PROPERTY xMoverPathFree : BOOL
GET
xMoverPathFree := THIS^.fb_Pnp.xOUT_MoverFree OR THIS^.fb_Pnp.xOUT_Ready OR THIS^.fb_Pnp.xOUT_Done;
END_GET
END_PROPERTY

PROPERTY xMoverShouldLeave : BOOL
GET
xMoverShouldLeave := THIS^.fb_Pnp.iOUT_Step = ST120_Pnp_e.SYNC_MOVER_LEAVE;
END_GET
END_PROPERTY

END_FUNCTION_BLOCK

// ---- POUs/20_AUTO/ST120/FB_ABL_120_Pnp.TcPOU
FUNCTION_BLOCK FB_ABL_120_Pnp
(****************************************************************************************)
(*	TITEL				laden kristall- Modul	    										*)
(*	Status				ungetestet                         								*)
(*	Beschrieb:			Ablaufbeschreibung												*)
(*																						*)
(*	Steps:	self-explained using enum													*)
(***********************************Revisionen*******************************************)
(*	see github blames																	*)
(****************************************************************************************)

VAR_INPUT
    xIN_Reset       : BOOL;          // Schrittkette zurücksetzen 
    xIN_Init        : BOOL;          // Initialisieren
    xIN_Quit        : BOOL;          // Fehler quittieren 
    xIN_Start       : BOOL;          // Startbefehl
    xIN_Sperre      : BOOL;          // FB Sperren 
    xIN_NextStep    : BOOL;          // Nächsten Schritt ausführen 
    xIN_AlarmAktiv  : BOOL;          // Anlage hat Alarm
    xIN_DryCycle    : BOOL;          // Fahren ohne Teile
    xIN_RestartCYCL : BOOL;          // Zyklus erneut starten im STEP, END, LEERFAHREN
    enIN_State      : enState;       // Status Anlage
    tIN_Timeout     : TIME := T#10s; // Timout

    pxFG_Freigabe : POINTER TO BOOL; //Freigabe von Station

    // Application specific
    Mover              : REFERENCE TO FB_Mover;
    xIN_PceReadyToPick : BOOL; // the piece(s) is/are ready to picked
END_VAR
VAR_OUTPUT
    (* standart Ausgänge *)
    xOUT_ErrFlag  : BOOL;        // Error Flag 
    xOUT_Busy     : BOOL;        // Baustein befindet sich im Ablauf 
    xOUT_Done     : BOOL;        // Baustein hat den Ablauf beendet 		
    xOUT_Ready    : BOOL;        // Ready to begin, should be the same state as done	
    xOUT_Timeout  : BOOL;        // Timeout FB 
    xOUT_InitDone : BOOL;        // initialisierung fertig
    xOUT_Wait     : BOOL;        // Wartet auf Bedingung
    iOUT_Step     : ST120_Pnp_e; // Aktueller Schritt 
    sOUT_Step     : STRING;      // Aktueller Schritt but in string format
    bOUT_Error    : BYTE;        // Fehlernummer

    iOUT_ProcessCompletion : INT;  //process completion, express in % (0-100)
    xOUT_MoverFree         : BOOL; // The mover is free to move
    xOUT_PickPiece         : BOOL; // Set to true when a piece is picked

END_VAR
VAR
    (* Standard *)
    (* Schritt *)
    iLastStep : ST120_Pnp_e; // Merker letzter Schritt 
    iPreStep  : ST120_Pnp_e; // Schritt zurück nach Alarm 
    iAktStep  : ST120_Pnp_e; // aktueller Schritt

    // Trigger Starten 
    rtSTART : R_TRIG;
    // Timer TimeOut 
    TON_Timeout : TON;

    (* Bausteine *)

    (* Spezial *)
    fb_axis120_01Y : FB_AxisLM_V1_1;
    fb_axis120_02Z : FB_AxisLM_V1_1;

    fb_PnpHorAxis : FB_LinearMotionMan;
    fb_PnpVerAxis : FB_LinearMotionMan;

    fb_gripperLeft    : FB_ZylMo2El_V2_1;
    fb_gripperRight   : FB_ZylMo2El_V2_1;
    simu_gripperLeft  : FB_Simu_Zyl2Pos;
    simu_gripperRight : FB_Simu_Zyl2Pos;

    fb_simu_axis120_01Y : FB_Simu_AxisLM_V1_1;
    fb_simu_axis120_02Z : FB_Simu_AxisLM_V1_1;

END_VAR
VAR CONSTANT
    PNP_SIMULATION : BOOL := FALSE; // Set to TRUE to simulate this part of the program
END_VAR

(*******************************************************************)
(* Trigger  *)
(*******************************************************************)
(* Zurücksetzen *)
IF xIN_RESET THEN
    iPreStep  := ST120_Pnp_e.RESET;
    iOUT_Step := ST120_Pnp_e.RESET;
END_IF

(* Error Quittieren *)
IF (bOUT_Error <> 0) AND xIN_Quit THEN
    xOUT_ErrFlag := FALSE;
    bOUT_Error   := 0;
    iOUT_Step    := iPreStep;
END_IF

(*******************************************************************)
(* Timer *)
(*******************************************************************)
TON_Timeout(IN := xIN_NextStep AND (iLastStep = iOUT_Step) (*todo FG *) ,
            PT := tIN_Timeout);

(*******************************************************************)
(* Bausteine *)
(*******************************************************************)
fb_PnpHorAxis(config          := _20_AUTO.recipe.linearAxis[LinearAxis_e.ST120_01Y],
              xIN_Init        := enIN_State = enState.StateINIT,
              xIN_Reset       := xIN_Reset,
              lrIN_CurrPos    := fb_axis120_01Y.rOUT_ActPos,
              lrIN_Delta_mm   := 0.5,
              iIN_CurrentStep := iOUT_Step,
              iIN_moveNumber  := ST120_PnpHorPos_e._max);

fb_simu_axis120_01Y(xIN_Enable          := PNP_SIMULATION AND CONST.USE_SIMULATION,
                    bIN_AxisCntr        := fb_axis120_01Y.bOUT_AxisCntr,
                    wIN_AxisState       := ST120_Axis.axis120_01Y.wState,
                    udiIN_HomingTime_ms := 2000,
                    pIN_axisSimu        := ADR(SIMU.axis_ref[Axis_e.ST120_01Y]),
                    pIN_axisHW          := ADR(ST120_Axis.axis120_01Y.axis),
                    rIN_PosActual       := fb_axis120_01Y.rOUT_ActPos,
                    rIN_PosMax          := ST120_Axis.const120_01Y.POS_MAX,
                    rIN_PosMin          := ST120_Axis.const120_01Y.POS_MIN,
                    rIN_PixMax          := 100,
                    rIN_PixMin          := 0);

fb_axis120_01Y(enIN_State       := enIN_State,
               parIN_Buttons    := ADR(AXIS.btTeachArAxis[Axis_e.ST120_01Y]),
               xIN_DisButtons   :=,
               xIN_Quit         := xIN_Quit,
               xIN_PARAMok      := TRUE, (*TODO*)
               xIN_FREE         := TRUE,
               xIN_FREE_HOME    := TRUE,
               rIN_POSMIN       := ST120_Axis.const120_01Y.POS_MIN,
               rIN_POSMAX       := ST120_Axis.const120_01Y.POS_MAX,
               rIN_VELOMAX      := ST120_Axis.const120_01Y.VELO_MAX,
               rIN_VELOMANU     := ST120_Axis.const120_01Y.VELO_MANU,
               rIN_VELOOPEN     := ST120_Axis.const120_01Y.VELO_MANU / 4,
               rIN_JogInc       := AXIS.rTeachIncAxis,
               xIN_Execute      := fb_PnpHorAxis.xOUT_Execute,
               xIN_Home         := ST120_Pnp_e.Init_HomeHorizontals = iAktStep,
               xIN_Relative     :=,
               rIN_Position     := TO_REAL(fb_PnpHorAxis.OUT_MoveProfile.lrPosition),
               rIN_Velocity     := TO_REAL(fb_PnpHorAxis.OUT_MoveProfile.lrVelocity),
               rIN_Acceleration := TO_REAL(fb_PnpHorAxis.OUT_MoveProfile.lrAccel),
               rIN_Deceleration := TO_REAL(fb_PnpHorAxis.OUT_MoveProfile.lrDecel),
               rIN_Jerk         := TO_REAL(fb_PnpHorAxis.OUT_MoveProfile.lrJerk),
               rIN_PosManu      :=
               TO_REAL(_20_AUTO.recipe
                           .linearAxis[LinearAxis_e.ST120_01Y].movesList[AXIS.bTeachPos[Axis_e.ST120_01Y]].lrPosition),
               rIN_VeloJogManu := TO_REAL(Axis.rJogVelo_pc),
               xIN_Reset       := (ST120_Pnp_e.RESET = iAktStep) OR xIN_Reset,
               // the simu fb gives the hardware signal when the simulation is disabled
               wAxisState    := fb_simu_axis120_01Y.wOUT_AxisState,
               bOUT_AxisCntr => ST120_Axis.axis120_01Y.bCtrlHi,
               rOUT_ActPos   => ST120_Axis.axis120_01Y.rActPos,
               axisIN_REF    := fb_simu_axis120_01Y.pOUT_axisRef^);

fb_PnpVerAxis(config          := _20_AUTO.recipe.linearAxis[LinearAxis_e.ST120_02Z],
              xIN_Init        := enIN_State = enState.StateINIT,
              xIN_Reset       := xIN_Reset,
              lrIN_CurrPos    := fb_axis120_02Z.rOUT_ActPos,
              lrIN_Delta_mm   := 0.5,
              iIN_CurrentStep := iOUT_Step,
              iIN_moveNumber  := ST120_PnpVerPos_e._max);

fb_simu_axis120_02Z(xIN_Enable          := PNP_SIMULATION AND CONST.USE_SIMULATION,
                    bIN_AxisCntr        := fb_axis120_02Z.bOUT_AxisCntr,
                    wIN_AxisState       := ST120_Axis.axis120_02Z.wState,
                    udiIN_HomingTime_ms := 2000,
                    pIN_axisSimu        := ADR(SIMU.axis_ref[Axis_e.ST120_02Z]),
                    pIN_axisHW          := ADR(ST120_Axis.axis120_02Z.axis),
                    rIN_PosActual       := fb_axis120_02Z.rOUT_ActPos,
                    rIN_PosMax          := ST120_Axis.const120_02Z.POS_MAX,
                    rIN_PosMin          := ST120_Axis.const120_02Z.POS_MIN,
                    rIN_PixMax          := 100,
                    rIN_PixMin          := 0);

fb_axis120_02Z(enIN_State       := enIN_State,
               parIN_Buttons    := ADR(AXIS.btTeachArAxis[Axis_e.ST120_02Z]),
               xIN_DisButtons   :=,
               xIN_Quit         := xIN_Quit,
               xIN_PARAMok      := TRUE, (*TODO*)
               xIN_FREE         := TRUE,
               xIN_FREE_HOME    := TRUE,
               rIN_POSMIN       := ST120_Axis.const120_02Z.POS_MIN,
               rIN_POSMAX       := ST120_Axis.const120_02Z.POS_MAX,
               rIN_VELOMAX      := ST120_Axis.const120_02Z.VELO_MAX,
               rIN_VELOMANU     := ST120_Axis.const120_02Z.VELO_MANU,
               rIN_VELOOPEN     := ST120_Axis.const120_02Z.VELO_MANU / 4,
               rIN_JogInc       := AXIS.rTeachIncAxis,
               xIN_Execute      := fb_PnpVerAxis.xOUT_Execute,
               xIN_Home         := ST120_Pnp_e.Init_HomeVerticals = iAktStep,
               xIN_Relative     :=,
               rIN_Position     := TO_REAL(fb_PnpVerAxis.OUT_MoveProfile.lrPosition),
               rIN_Velocity     := TO_REAL(fb_PnpVerAxis.OUT_MoveProfile.lrVelocity),
               rIN_Acceleration := TO_REAL(fb_PnpVerAxis.OUT_MoveProfile.lrAccel),
               rIN_Deceleration := TO_REAL(fb_PnpVerAxis.OUT_MoveProfile.lrDecel),
               rIN_Jerk         := TO_REAL(fb_PnpVerAxis.OUT_MoveProfile.lrJerk),
               rIN_PosManu      :=
               TO_REAL(_20_AUTO.recipe
                           .linearAxis[LinearAxis_e.ST120_02Z].movesList[AXIS.bTeachPos[Axis_e.ST120_02Z]].lrPosition),
               rIN_VeloJogManu := TO_REAL(Axis.rJogVelo_pc),
               xIN_Reset       := (ST120_Pnp_e.RESET = iAktStep) OR xIN_Reset,
               // the simu fb gives the hardware signal when the simulation is disabled
               wAxisState    := fb_simu_axis120_02Z.wOUT_AxisState,
               bOUT_AxisCntr => ST120_Axis.axis120_02Z.bCtrlHi,
               rOUT_ActPos   => ST120_Axis.axis120_02Z.rActPos,
               axisIN_REF    := fb_simu_axis120_02Z.pOUT_axisRef^);

fb_gripperLeft(xIN_Reset    := xIN_Reset OR (ST120_Pnp_e.RESET = iOUT_Step),
               xIN_Quit     := xIN_Quit,
               xIN_Manu     := enState.StateMANU = enIN_State,
               pbtIN_Button := ADR(HMI.btManuCylinders[StationList_e.ST120][1]),
               xIN_GS       := simu_gripperLeft.xOUT_inGS,
               xIN_AS       := simu_gripperLeft.xOUT_inAS,
               xIN_FREE     := TRUE,
               xINtoGS      := (ST120_Pnp_e.Gripper_open = iOUT_Step) OR
                               (ST120_Pnp_e.Init_open_left_clamp = iOUT_Step),
               xINtoAS      := _20_AUTO.recipe.st120.xUseVerLeft AND ST120_Pnp_e.Gripper_close = iOUT_Step,
               tIN_ErrAS := DINT_TO_TIME(_20_AUTO.recipe.cylinder2Pos[StationList_e.ST120]
                                             [ST120_Cylinders_e.GreiferLinks].toAS_alarm_time),
               tIN_ErrGS := DINT_TO_TIME(_20_AUTO.recipe.cylinder2Pos[StationList_e.ST120]
                                             [ST120_Cylinders_e.GreiferLinks].toGS_alarm_time),
               tIN_WaitAS := DINT_TO_TIME(_20_AUTO.recipe.cylinder2Pos[StationList_e.ST120]
                                              [ST120_Cylinders_e.GreiferLinks].toAS_wait_time),
               tIN_WaitGS := DINT_TO_TIME(_20_AUTO.recipe.cylinder2Pos[StationList_e.ST120]
                                              [ST120_Cylinders_e.GreiferLinks].toGS_wait_time));

simu_gripperLeft(xIN_Enable := TRUE, // PNP_SIMULATION AND CONST.USE_SIMULATION,
                 xIN_inGS   := IO_BOX.I6300_ST120_greifer_links_geschlossen,
                 xIN_inAS   := IO_BOX.I6301_ST120_greifer_links_offen,
                 xIN_valve  := fb_gripperLeft.xOUT_VALVE,
                 tIN_GS_ms  := 200,  //ms
                 tIN_AS_ms  := 200); //ms

fb_gripperRight(xIN_Reset    := xIN_Reset OR (ST120_Pnp_e.RESET = iOUT_Step),
                xIN_Quit     := xIN_Quit,
                xIN_Manu     := enState.StateMANU = enIN_State,
                pbtIN_Button := ADR(HMI.btManuCylinders[StationList_e.ST120][2]),
                xIN_GS       := simu_gripperRight.xOUT_inGS,
                xIN_AS       := simu_gripperRight.xOUT_inAS,
                xIN_FREE     := TRUE,
                xINtoGS      := (ST120_Pnp_e.Gripper_open = iOUT_Step) OR
                                (ST120_Pnp_e.Init_open_right_clamp = iOUT_Step),
                xINtoAS      := _20_AUTO.recipe.st120.xUseVerRight AND (ST120_Pnp_e.Gripper_close = iOUT_Step),
                tIN_ErrAS := DINT_TO_TIME(_20_AUTO.recipe.cylinder2Pos[StationList_e.ST120]
                                              [ST120_Cylinders_e.GreiferRechts].toAS_alarm_time),
                tIN_ErrGS := DINT_TO_TIME(_20_AUTO.recipe.cylinder2Pos[StationList_e.ST120]
                                              [ST120_Cylinders_e.GreiferRechts].toGS_alarm_time),
                tIN_WaitAS := DINT_TO_TIME(_20_AUTO.recipe.cylinder2Pos[StationList_e.ST120]
                                               [ST120_Cylinders_e.GreiferRechts].toAS_wait_time),
                tIN_WaitGS := DINT_TO_TIME(_20_AUTO.recipe.cylinder2Pos[StationList_e.ST120]
                                               [ST120_Cylinders_e.GreiferRechts].toGS_wait_time));

simu_gripperRight(xIN_Enable := TRUE, // PNP_SIMULATION AND CONST.USE_SIMULATION,
                  xIN_inGS   := IO_BOX.I6302_ST120_greifer_rechts_geschlossen,
                  xIN_inAS   := IO_BOX.I6303_ST120_greifer_rechts_offen,
                  xIN_valve  := fb_gripperRight.xOUT_VALVE,
                  tIN_GS_ms  := 200,  //ms
                  tIN_AS_ms  := 200); //ms

(*******************************************************************)
(* OUTPUTS *)
(*******************************************************************)
// Error Flag 
xOUT_ErrFlag := (bOUT_Error <> 0) OR (ST120_Pnp_e.ERROR = iOUT_Step);
// Baustein befindet sich im Ablauf 
xOUT_Busy := (iOUT_Step > ST120_Pnp_e.READY) AND (iOUT_Step < ST120_Pnp_e.DONE);
// Baustein hat den Ablauf beendet
xOUT_Done := (iOUT_Step = ST120_Pnp_e.DONE);
// Process ready
xOUT_Ready := (iOUT_Step = ST120_Pnp_e.READY) OR (iOUT_Step = ST120_Pnp_e.waitOnMover);
// Timeout FB 				 		
xOUT_Timeout := TON_Timeout.Q;
// Itialisierung fertig			
xOUT_InitDone := (iOUT_Step = ST120_Pnp_e.READY) OR (iOUT_Step = ST120_Pnp_e.waitOnMover);
// Aktueller Schritt			
iOUT_Step := iOUT_Step; //Im Ablauf gesetzt		
sOUT_Step := TO_STRING(iOUT_Step);
//Fehlernummer	 
bOUT_Error := bOUT_Error; //Im Ablauf/FB gesetzt	
(* Warte (alle Schritte wo auf FG oder Teile gewartet wird) *)
xOUT_Wait := (iOUT_Step = ST120_Pnp_e.DONE) OR
             (iOUT_Step = ST120_Pnp_e.READY) OR
             (iOUT_Step = ST120_Pnp_e.START) OR
             (iOUT_Step = ST120_Pnp_e.waitOnMover) OR
             (iOUT_Step = ST120_Pnp_e.SYNC_MOVER_LEAVE) OR
             (iOUT_Step = ST120_Pnp_e.PnP_WaitOnFeeder);

xOUT_MoverFree := iOUT_Step >= ST120_Pnp_e.MOVER_FREE_OP AND iOUT_Step < ST120_Pnp_e.MOVER_NEEDED_OP;

iOUT_ProcessCompletion := F_GetPercent_2(iAktStep,
                                         ST120_Pnp_e.PnP_Hor_ToRotTablePos,
                                         ST120_Pnp_e.PnP_Hor_ToTrackPos,
                                         ST120_Pnp_e.PnP_Ver_ShuttleDown,
                                         ST120_Pnp_e.PnP_Ver_ShuttleUp);

xOUT_PickPiece := iOUT_Step = ST120_Pnp_e.PnP_Ver_RotTableUp;

IO_BOX.Q5202_14_ST120_greifer_links  := fb_gripperLeft.xOUT_VALVE AND NOT (PNP_SIMULATION AND CONST.USE_SIMULATION);
IO_BOX.Q5203_14_ST120_greifer_rechts := fb_gripperRight.xOUT_VALVE AND NOT (PNP_SIMULATION AND CONST.USE_SIMULATION);

IO_BOX.Q5212_14_ST120_stop_vertical_axis := NOT fb_simu_axis120_02Z.pIN_axisHW^.Status.Error AND
                                            _02_SAFETY.xOUT_ESout AND
                                            _02_SAFETY.xOUT_MonOut AND
                                            NOT (PNP_SIMULATION AND CONST.USE_SIMULATION);

(*******************************************************************)
(* Ablauf *)
(*******************************************************************)

(* Sperren *)
IF xIN_Sperre THEN
    iPreStep  := ST120_Pnp_e.RESET;
    iOUT_Step := ST120_Pnp_e.RESET;
    RETURN;
END_IF;

(* Schritt Merker *)
IF iAktStep <> iOUT_Step THEN
    iLastStep := iAktStep;
    iAktStep  := iOUT_Step;
END_IF

(* START *)
rtSTART(CLK := xIN_Start);

IF 0 = bOUT_Error THEN
    IF fb_axis120_01Y.xOUT_ErrFlag THEN
        bOUT_Error := ST120_Alarm_e.Axis_120_01Y_error;
    ELSIF fb_axis120_02Z.xOUT_ErrFlag THEN
        bOUT_Error := ST120_Alarm_e.Axis_120_02Z_error;
    ELSIF fb_gripperLeft.xOUT_ErrFlag THEN
        bOUT_Error := ST120_Alarm_e.Cylinder_griper_left;
    ELSIF fb_gripperRight.xOUT_ErrFlag THEN
        bOUT_Error := ST120_Alarm_e.Cylinder_griper_right;
    END_IF
ELSIF iOUT_Step < ST120_Pnp_e.ERROR THEN
    iOUT_Step := ST120_Pnp_e.ERROR;
END_IF

(*******************************************************************)
(* Schrittkette  *)
(*******************************************************************)
CASE iOUT_Step OF

(***** RESET *****)
ST120_Pnp_e.RESET: (* Schritt 0-99 *)
    //Initialisierungen
    //Start Init Ablauf
    IF xIN_Init THEN
        iOUT_Step := ST120_Pnp_e.INIT;
        //Start Manu Ablauf
    ELSIF enIN_State = StateMANU AND xIN_NextStep THEN
        iOUT_Step := ST120_Pnp_e.INIT;
    END_IF;

(***** INIT *****)
ST120_Pnp_e.INIT: (* Grundstellung ? *)
    IF fb_axis120_02Z.xOUT_HOMED THEN
        iOUT_Step := ST120_Pnp_e.Init_VerticalsUp;
    ELSE
        iOUT_Step := ST120_Pnp_e.Init_HomeVerticals;
    END_IF

ST120_Pnp_e.Init_HomeVerticals:
    IF fb_axis120_02Z.xOUT_HOMED THEN
        iOUT_Step := ST120_Pnp_e.Init_VerticalsUp;
    END_IF

ST120_Pnp_e.Init_VerticalsUp:
    IF fb_gripperLeft.xIN_AS OR fb_gripperRight.xIN_AS THEN
        IF fb_PnpVerAxis.MoveTo(ST120_PnpVerPos_e.UpFull).xOUT_InPos THEN
            IF fb_axis120_01Y.xOUT_READY OR fb_axis120_01Y.xOUT_HOMED THEN
                iOUT_Step := ST120_Pnp_e.Init_HorizontalsToTrack;
            ELSE
                iOUT_Step := ST120_Pnp_e.Init_HomeHorizontals;
            END_IF
        END_IF
    ELSE
        IF fb_PnpVerAxis.MoveTo(ST120_PnpVerPos_e.UpEmpty).xOUT_InPos THEN
            IF fb_axis120_01Y.xOUT_READY OR fb_axis120_01Y.xOUT_HOMED THEN
                iOUT_Step := ST120_Pnp_e.Init_HorizontalsToTrack;
            ELSE
                iOUT_Step := ST120_Pnp_e.Init_HomeHorizontals;
            END_IF
        END_IF
    END_IF

ST120_Pnp_e.Init_HomeHorizontals:
    IF fb_axis120_01Y.xOUT_HOMED THEN
        iOUT_Step := ST120_Pnp_e.Init_HorizontalsToTrack;
    END_IF

ST120_Pnp_e.Init_HorizontalsToTrack:
    IF fb_PnpHorAxis.MoveTo(ST120_PnpHorPos_e.GS).xOUT_InPos THEN
        iOUT_Step := ST120_Pnp_e.Init_adjust_left_clamp;
    END_IF

ST120_Pnp_e.Init_adjust_left_clamp:
    // a piece is in the griper when there is no GS signal
    IF _20_AUTO.recipe.st120.xUseVerLeft THEN
        iOUT_Step := ST120_Pnp_e.Init_adjust_right_clamp;
    ELSE
        iOUT_Step := ST120_Pnp_e.Init_open_left_clamp;
    END_IF

ST120_Pnp_e.Init_open_left_clamp:
    IF fb_gripperLeft.xIN_GS THEN
        IF _20_AUTO.recipe.st120.xUseVerRight THEN
            iOUT_Step := ST120_Pnp_e.Init_adjust_right_clamp;
        ELSE
            iOUT_Step := ST120_Pnp_e.Init_check_if_pces_handled;
        END_IF
    END_IF

ST120_Pnp_e.Init_adjust_right_clamp:
    // a piece is in the griper when there is no GS signal
    IF _20_AUTO.recipe.st120.xUseVerRight THEN
        iOUT_Step := ST120_Pnp_e.Init_check_if_pces_handled;
    ELSE
        iOUT_Step := ST120_Pnp_e.Init_open_right_clamp;
    END_IF

ST120_Pnp_e.Init_open_right_clamp:
    IF fb_gripperRight.xIN_GS THEN
        iOUT_Step := ST120_Pnp_e.Init_check_if_pces_handled;
    END_IF

ST120_Pnp_e.Init_check_if_pces_handled:
    IF (NOT _20_AUTO.recipe.st120.xUseVerLeft AND NOT fb_gripperLeft.xIN_GS) OR
       (NOT _20_AUTO.recipe.st120.xUseVerRight AND NOT fb_gripperRight.xIN_GS) THEN
        bOUT_Error := ST120_Alarm_e.Piece_in_unused_griper;
        iOUT_Step  := ST120_Pnp_e.ERROR;

    ELSIF (_20_AUTO.recipe.st120.xUseVerLeft AND fb_gripperLeft.xIN_GS) AND
          (_20_AUTO.recipe.st120.xUseVerRight AND NOT fb_gripperRight.xIN_GS) THEN
        bOUT_Error := ST120_Alarm_e.Piece_missing_left_griper;
        iOUT_Step  := ST120_Pnp_e.ERROR;

    ELSIF (_20_AUTO.recipe.st120.xUseVerLeft AND NOT fb_gripperLeft.xIN_GS) AND
          (_20_AUTO.recipe.st120.xUseVerRight AND fb_gripperRight.xIN_GS) THEN
        bOUT_Error := ST120_Alarm_e.Piece_missing_right_griper;
        iOUT_Step  := ST120_Pnp_e.ERROR;

        // if both are open, we don't make further checks
    ELSIF (NOT _20_AUTO.recipe.st120.xUseVerLeft OR fb_gripperLeft.xOUT_inGS) AND
          (NOT _20_AUTO.recipe.st120.xUseVerRight OR fb_gripperRight.xOUT_inGS) THEN
        iOUT_Step := ST120_Pnp_e.waitOnMover;

    ELSE
        iOUT_Step := ST120_Pnp_e.READY;
    END_IF

(***** READY / INIT DONE *****)
ST120_Pnp_e.READY:    (* Start AUTO,END,LEER,STEP *)
    IF xIN_Start THEN //IF rtSTART.Q THEN
        iOUT_Step := ST120_Pnp_e.START;
    END_IF

(***** START  ZYKLISCH *****)
ST120_Pnp_e.START: (*  *)
    IF xIN_NextStep AND pxFG_Freigabe^ THEN
        IF enState.StateLEER = enIN_State THEN
            IF __ISVALIDREF(Mover) THEN
                IF Mover.GetLastStationDone() > 0 THEN
                    iOUT_Step := ST120_Pnp_e.PnP_Hor_ToRotTablePos;
                ELSE
                    iOUT_Step := ST120_Pnp_e.waitOnMover;
                END_IF
            END_IF
        ELSE
            iOUT_Step := ST120_Pnp_e.PnP_Hor_ToRotTablePos;
        END_IF
    END_IF;

ST120_Pnp_e.PnP_Hor_ToRotTablePos:
    IF xIN_NextStep AND fb_PnpHorAxis.MoveTo(ST120_PnpHorPos_e.AS).xOUT_InPos THEN
        iOUT_Step := ST120_Pnp_e.PnP_WaitOnFeeder;
    END_IF

ST120_Pnp_e.PnP_WaitOnFeeder:
    IF xIN_PceReadyToPick THEN
        iOUT_Step := ST120_Pnp_e.PnP_Ver_RotTableDown;
    END_IF

ST120_Pnp_e.PnP_Ver_RotTableDown:
    IF xIN_NextStep AND fb_PnpVerAxis.MoveTo(ST120_PnpVerPos_e.DownEmpty).xOUT_InPos THEN
        iOUT_Step := ST120_Pnp_e.Gripper_close;
    END_IF;

ST120_Pnp_e.Gripper_close:
    IF xIN_NextStep AND
       (NOT _20_AUTO.recipe.st120.xUseVerLeft OR fb_gripperLeft.xOUT_inAS) AND
       (NOT _20_AUTO.recipe.st120.xUseVerRight OR fb_gripperRight.xOUT_inAS) THEN
        iOUT_Step := ST120_Pnp_e.PnP_Ver_RotTableUp;
    END_IF;

ST120_Pnp_e.PnP_Ver_RotTableUp:
    IF xIN_NextStep AND fb_PnpVerAxis.MoveTo(ST120_PnpVerPos_e.UpFull).xOUT_InPos THEN
        iOUT_Step := ST120_Pnp_e.PnP_Hor_ToTrackPos;
    END_IF;

ST120_Pnp_e.PnP_Hor_ToTrackPos:
    IF xIN_NextStep AND fb_PnpHorAxis.MoveTo(ST120_PnpHorPos_e.GS).xOUT_InPos THEN
        iOUT_Step := ST120_Pnp_e.waitOnMover;
    END_IF

ST120_Pnp_e.waitOnMover: (*  *)
    IF xIN_NextStep AND __ISVALIDREF(Mover) OR HMI.bArForceCyclusState[StationList_e.ST120] THEN
        IF Mover.GetLastStationDone() >= INT#120 THEN
            iOUT_Step := ST120_Pnp_e.SYNC_MOVER_LEAVE;
        ELSIF Mover.GetLastStationDone() < INT#105 THEN
            iOUT_Step := ST120_Pnp_e.SYNC_MOVER_LEAVE;
        ELSE
            iOUT_Step := ST120_Pnp_e.PnP_Ver_ShuttleDown;
        END_IF
    END_IF;

ST120_Pnp_e.PnP_Ver_ShuttleDown:
    IF xIN_NextStep AND fb_PnpVerAxis.MoveTo(ST120_PnpVerPos_e.DownFullQuick).xOUT_InPos THEN
        iOUT_Step := ST120_Pnp_e.PnP_Ver_ShuttleTorqueControl;

        IF __ISVALIDREF(Mover) THEN
            IF NOT Mover.SetLastStation(120) THEN
                ASSERT(0);
            END_IF
        END_IF
    END_IF;

// We need a fb that enables for us torque control. Here we just go a bit further
ST120_Pnp_e.PnP_Ver_ShuttleTorqueControl:
    IF xIN_NextStep AND fb_PnpVerAxis.MoveTo(ST120_PnpVerPos_e.DownFullTorqueControl).xOUT_InPos THEN
        iOUT_Step := ST120_Pnp_e.Gripper_open;
    END_IF;

ST120_Pnp_e.Gripper_open:
    IF xIN_NextStep AND
       (NOT _20_AUTO.recipe.st120.xUseVerLeft OR fb_gripperLeft.xOUT_inGS) AND
       (NOT _20_AUTO.recipe.st120.xUseVerRight OR fb_gripperRight.xOUT_inGS) THEN
        iOUT_Step := ST120_Pnp_e.PnP_Ver_ShuttleUp;
    END_IF;

ST120_Pnp_e.PnP_Ver_ShuttleUp:
    IF xIN_NextStep AND fb_PnpVerAxis.MoveTo(ST120_PnpVerPos_e.UpEmpty).xOUT_InPos THEN
        iOUT_Step := ST120_Pnp_e.SYNC_MOVER_LEAVE;

        IF __ISVALIDREF(Mover) THEN
            IF NOT Mover.SetLastStation(120) THEN
                ASSERT(0);
            END_IF
        END_IF
    END_IF;

ST120_Pnp_e.SYNC_MOVER_LEAVE:
    // The mover needs to be taken by MoverMan
    IF NOT __ISVALIDREF(Mover) THEN
        IF (NOT _20_AUTO.recipe.st120.xUseVerLeft OR fb_gripperLeft.xOUT_inGS AND
           (NOT _20_AUTO.recipe.st120.xUseVerRight OR fb_gripperRight.xOUT_inGS) THEN
            iOUT_Step := ST120_Pnp_e.DONE;
        ELSE
            iOUT_Step := ST120_Pnp_e.waitOnMover;
        END_IF
    END_IF

(***** DONE *****)
ST120_Pnp_e.DONE: (* Letzter Schritt  *)
    IF NOT xIN_AlarmAktiv THEN
        //AUTO
        IF (enIN_State = StateAUTO) AND xIN_RestartCYCL THEN
            iOUT_Step := ST120_Pnp_e.START;
            //STEP / END / LEERFAHREN restart
        ELSIF (enIN_State < StateAUTO) AND (enIN_State >= enState.StateSTEP) AND xIN_RestartCYCL THEN
            iOUT_Step := ST120_Pnp_e.START;
            //STEP / END / LEERFAHREN fertig
        ELSIF (enIN_State = StateREADY) THEN
            iOUT_Step := ST120_Pnp_e.READY;
        END_IF;
    END_IF;

(************ ERROR *************)
ST120_Pnp_e.ERROR: (* ERROR *) ;

END_CASE;

END_FUNCTION_BLOCK

// ---- POUs/20_AUTO/ST120/FB_ABL_120_Feeder.TcPOU
FUNCTION_BLOCK FB_ABL_120_Feeder
(****************************************************************************************)
(*	TITEL				laden Kristall modul, Feeder and rotary table                   *)
(*	Status				ungetestet                         								*)
(*	Beschrieb:			Ablaufbeschreibung												*)
(*																						*)
(*	Steps:	self-explained using enum													*)
(***********************************Revisionen*******************************************)
(*	see github blames																	*)
(****************************************************************************************)

VAR_INPUT
    xIN_Reset       : BOOL;          // Schrittkette zurücksetzen 
    xIN_Init        : BOOL;          // Initialisieren
    xIN_Quit        : BOOL;          // Fehler quittieren 
    xIN_Start       : BOOL;          // Startbefehl
    xIN_Sperre      : BOOL;          // FB Sperren 
    xIN_NextStep    : BOOL;          // Nächsten Schritt ausführen 
    xIN_AlarmAktiv  : BOOL;          // Anlage hat Alarm
    xIN_DryCycle    : BOOL;          // Fahren ohne Teile
    xIN_RestartCYCL : BOOL;          // Zyklus erneut starten im STEP, END, LEERFAHREN
    enIN_State      : enState;       // Status Anlage
    tIN_Timeout     : TIME := T#10s; // Timout

    pxFG_Freigabe : POINTER TO BOOL; //Freigabe von Station

    // Application specific
    xIN_PickPiece : BOOL; (* signal from the pick and place element
                             the number of picked signal depend on the recipe *)
    xIN_PnpGripperOpen : BOOL; // the gripper of the pnp part is open
    xIN_PnpNotOnTheWay : BOOL; // the pnp is at the track side or up enough
END_VAR
VAR_OUTPUT
    (* standart Ausgänge *)
    xOUT_ErrFlag  : BOOL;           // Error Flag 
    xOUT_Busy     : BOOL;           // Baustein befindet sich im Ablauf 
    xOUT_Done     : BOOL;           // Baustein hat den Ablauf beendet 		
    xOUT_Ready    : BOOL;           // Ready to begin, should be the same state as done	
    xOUT_Timeout  : BOOL;           // Timeout FB 
    xOUT_InitDone : BOOL;           // initialisierung fertig
    xOUT_Wait     : BOOL;           // Wartet auf Bedingung
    iOUT_Step     : ST120_Feeder_e; // Aktueller Schritt 
    sOUT_Step     : STRING;         // Aktueller Schritt but in string format
    bOUT_Error    : BYTE;           // Fehlernummer

    // Application specific
    xOUT_PceReadyToPick : BOOL; // the piece(s) is/are ready to picked
END_VAR
VAR
    (* Standard *)
    (* Schritt *)
    iLastStep : ST120_Feeder_e; // Merker letzter Schritt 
    iPreStep  : ST120_Feeder_e; // Schritt zurück nach Alarm 
    iAktStep  : ST120_Feeder_e; // aktueller Schritt

    // Trigger Starten 
    rtSTART : R_TRIG;
    // Timer TimeOut 
    TON_Timeout : TON;

    (* Bausteine *)
	btfb_feederLeft					: FB_BUTTON;
	btfb_feederRight				: FB_BUTTON;

    // Application specific^
    fb_pivotLeft    : FB_ZylMo2El_V2_1;
    fb_pivotRight   : FB_ZylMo2El_V2_1;
    simu_pivotLeft  : FB_Simu_Zyl2Pos;
    simu_pivotRight : FB_Simu_Zyl2Pos;

    simu_feederLeft  : FB_Simu_Feeder;                    // simulation of a feeder
    simu_feederRight : FB_Simu_Feeder;                    // simulation of a feeder
    simu_fifoLeft    : FB_Fifo(BAND_SIZE_FOR_TUBE_LEFT);  // fifo to hold a piece
    simu_fifoRight   : FB_Fifo(BAND_SIZE_FOR_TUBE_RIGHT); // fifo to hold a piece
    rtPutPieceLeft   : R_TRIG;                            // trigger to add a piece
    rtPutPieceRight  : R_TRIG;                            // trigger to add a piece

    fb_feederLeft      : FB_Feeder2Sensors;
    fb_feederRight     : FB_Feeder2Sensors;
    fb_hubladerLeft    : FB_ZylMo2El_V2_1;
    fb_hubladerRight   : FB_ZylMo2El_V2_1;
    simu_hubladerLeft  : FB_Simu_Zyl2Pos;
    simu_hubladerRight : FB_Simu_Zyl2Pos;

    simu_start_tick : UDINT; // simulation start tick, used to simulate movement

    TON_PieceInPivotLeft  : TON;
    TON_PieceInPivotRight : TON;

END_VAR
VAR CONSTANT
    BAND_SIZE_FOR_TUBE_LEFT  : INT := 3; // Band size, we assume that tubes pushe each other in order to move to the PNP machine
    BAND_SIZE_FOR_TUBE_RIGHT : INT := 2; // Band size, we assume that tubes pushe each other in order to move to the PNP machine

    FEEDER_SIMULATION : BOOL := FALSE; // Simulate this code
END_VAR

(*******************************************************************)
(* Trigger  *)
(*******************************************************************)
(* Zurücksetzen *)
IF xIN_RESET THEN
    iPreStep  := ST120_Feeder_e.RESET;
    iOUT_Step := ST120_Feeder_e.RESET;
END_IF;

(* Error Quittieren *)
IF (bOUT_Error <> 0) AND xIN_Quit THEN
    xOUT_ErrFlag := FALSE;
    bOUT_Error   := 0;
    iOUT_Step    := iPreStep;
END_IF;

(*******************************************************************)
(* Timer *)
(*******************************************************************)
TON_Timeout(IN := xIN_NextStep AND (iLastStep = iOUT_Step) (*todo FG *) ,
            PT := tIN_Timeout);

TON_PieceInPivotLeft(IN := IO_BOX.I6404_ST120_teil_in_vereizelung_links,
                     PT := DINT_TO_TIME(_20_AUTO.recipe.st120.TON_PieceInSeperatorLeft));

TON_PieceInPivotRight(IN := IO_BOX.I6405_ST120_teil_in_vereinzelung_rechts,
                      PT := DINT_TO_TIME(_20_AUTO.recipe.st120.TON_PieceInSeperatorRight));

(*******************************************************************)
(* Bausteine *)
(*******************************************************************)
fb_pivotLeft(xIN_Reset    := xIN_Reset OR (ST120_Feeder_e.RESET = iOUT_Step),
             xIN_Quit     := xIN_Quit,
             xIN_Manu     := enState.StateMANU = enIN_State,
             pbtIN_Button := ADR(HMI.btManuCylinders[StationList_e.ST120][3]),
             xIN_GS       := simu_pivotLeft.xOUT_inGS,
             xIN_AS       := simu_pivotLeft.xOUT_inAS,
             xIN_FREE     := xIN_PnpNotOnTheWay OR xIN_PnpGripperOpen,
             xINtoGS      :=
                 _20_AUTO.recipe.st120.xUseVerLeft AND
                 ((ST120_Feeder_e.rotate_to_pnp = iOUT_Step) OR (ST120_Feeder_e.Init_pivot_to_pnp = iOUT_Step)),
             xINtoAS := _20_AUTO.recipe.st120.xUseVerLeft AND
                        (ST120_Feeder_e.rotate_to_feeder = iOUT_Step OR
                        ST120_Feeder_e.Init_pivot_to_feeder = iOUT_Step),
             tIN_ErrAS := DINT_TO_TIME(_20_AUTO.recipe.cylinder2Pos[StationList_e.ST120]
                                           [ST120_Cylinders_e.GreiferLinks].toAS_alarm_time),
             tIN_ErrGS := DINT_TO_TIME(_20_AUTO.recipe.cylinder2Pos[StationList_e.ST120]
                                           [ST120_Cylinders_e.GreiferLinks].toGS_alarm_time),
             tIN_WaitAS := DINT_TO_TIME(_20_AUTO.recipe.cylinder2Pos[StationList_e.ST120]
                                            [ST120_Cylinders_e.GreiferLinks].toAS_wait_time),
             tIN_WaitGS := DINT_TO_TIME(_20_AUTO.recipe.cylinder2Pos[StationList_e.ST120]
                                            [ST120_Cylinders_e.GreiferLinks].toGS_wait_time));

simu_pivotLeft(xIN_Enable := FEEDER_SIMULATION AND CONST.USE_SIMULATION,
               xIN_inGS   := IO_BOX.I6400_ST120_schwenken_links_in_vertikal,
               xIN_inAS   := IO_BOX.I6401_ST120_schwenken_links_in_horizontal,
               xIN_valve  := fb_pivotLeft.xOUT_VALVE,
               tIN_GS_ms  := 500,  //ms
               tIN_AS_ms  := 500); //ms

fb_pivotRight(xIN_Reset    := xIN_Reset OR (ST120_Feeder_e.RESET = iOUT_Step),
              xIN_Quit     := xIN_Quit,
              xIN_Manu     := enState.StateMANU = enIN_State,
              pbtIN_Button := ADR(HMI.btManuCylinders[StationList_e.ST120][4]),
              xIN_GS       := simu_pivotRight.xOUT_inGS,
              xIN_AS       := simu_pivotRight.xOUT_inAS,
              xIN_FREE     := xIN_PnpGripperOpen OR xIN_PnpNotOnTheWay,
              xINtoGS      :=
                  _20_AUTO.recipe.st120.xUseVerRight AND
                  ((ST120_Feeder_e.rotate_to_pnp = iOUT_Step) OR (ST120_Feeder_e.Init_pivot_to_pnp = iOUT_Step)),
              xINtoAS := _20_AUTO.recipe.st120.xUseVerRight AND
                         (ST120_Feeder_e.rotate_to_feeder = iOUT_Step OR
                         ST120_Feeder_e.Init_pivot_to_feeder = iOUT_Step),
              tIN_ErrAS := DINT_TO_TIME(_20_AUTO.recipe.cylinder2Pos[StationList_e.ST120]
                                            [ST120_Cylinders_e.GreiferRechts].toAS_alarm_time),
              tIN_ErrGS := DINT_TO_TIME(_20_AUTO.recipe.cylinder2Pos[StationList_e.ST120]
                                            [ST120_Cylinders_e.GreiferRechts].toGS_alarm_time),
              tIN_WaitAS := DINT_TO_TIME(_20_AUTO.recipe.cylinder2Pos[StationList_e.ST120]
                                             [ST120_Cylinders_e.GreiferRechts].toAS_wait_time),
              tIN_WaitGS := DINT_TO_TIME(_20_AUTO.recipe.cylinder2Pos[StationList_e.ST120]
                                             [ST120_Cylinders_e.GreiferRechts].toGS_wait_time));

simu_pivotRight(xIN_Enable := FEEDER_SIMULATION AND CONST.USE_SIMULATION,
                xIN_inGS   := IO_BOX.I6402_ST120_schwenken_rechts_in_vertikal,
                xIN_inAS   := IO_BOX.I6403_ST120_schwenken_rechts_in_horizontal,
                xIN_valve  := fb_pivotRight.xOUT_VALVE,
                tIN_GS_ms  := 500,  //ms
                tIN_AS_ms  := 500); //ms

btfb_feederLeft(pbtIN  := ADR(HMI.btManuCylinders[StationList_e.ST120][7]),
                xINdis := (enIN_State <> enState.StateMANU),
                xINon  :=,
                xINerr := fb_feederLeft.xOUT_Empty);

IF btfb_feederLeft.pbtIN^.rtrig THEN
    btfb_feederLeft.xINon := NOT btfb_feederLeft.xINon;
ELSIF (enIN_State <> enState.StateMANU) THEN
    btfb_feederLeft.xINon := FALSE;
END_IF;

fb_feederLeft(xIN_Enable := (enIN_State = enState.StateAUTO OR enIN_State = enState.StateSTEP) AND
                            _20_AUTO.recipe.st120.xUseVerLeft,
              // here we do something special. We only want the hublader to run
              // when no piece are at the maxi sensor to prevent a stuck usage 
              xIN_PieceInEnd            := IO_BOX.I8304_ST120_maxi_zufurung_links,
              xIN_PieceMax              := IO_BOX.I8304_ST120_maxi_zufurung_links,
              xIN_InSimulation          := FEEDER_SIMULATION AND CONST.USE_SIMULATION,
              refIN_SimulatedFifo       := simu_fifoLeft,
              iIN_FifoSetMaxSensorValue := BAND_SIZE_FOR_TUBE_LEFT,
              diIN_SignlFilter_ms       := _20_AUTO.recipe.st120.FeederConfigLeft.InFilterDelay,
              diIN_StartDelay_ms        := _20_AUTO.recipe.st120.FeederConfigLeft.StartDelay,
              diIN_StopDelay_ms         := _20_AUTO.recipe.st120.FeederConfigLeft.StopDelay,
              diIN_EmptyDelay_ms        := _20_AUTO.recipe.st120.FeederConfigLeft.EmptyDelay);

btfb_feederRight(pbtIN  := ADR(HMI.btManuCylinders[StationList_e.ST120][8]),
                 xINdis := (enIN_State <> enState.StateMANU),
                 xINon  :=,
                 xINerr := fb_feederRight.xOUT_Empty);

IF btfb_feederRight.pbtIN^.rtrig THEN
    btfb_feederRight.xINon := NOT btfb_feederRight.xINon;
ELSIF (enIN_State <> enState.StateMANU) THEN
    btfb_feederRight.xINon := FALSE;
END_IF;

fb_feederRight(xIN_Enable := (enIN_State = enState.StateAUTO OR enIN_State = enState.StateSTEP) AND
                             _20_AUTO.recipe.st120.xUseVerRight,
               // here we do something special. We only want the hublader to run
               // when no piece are at the maxi sensor to prevent a stuck usage 
               xIN_PieceInEnd            := IO_BOX.I8305_ST120_maxi_zufurung_rechts,
               xIN_PieceMax              := IO_BOX.I8305_ST120_maxi_zufurung_rechts,
               xIN_InSimulation          := FEEDER_SIMULATION AND CONST.USE_SIMULATION,
               refIN_SimulatedFifo       := simu_fifoRight,
               iIN_FifoSetMaxSensorValue := BAND_SIZE_FOR_TUBE_RIGHT,
               diIN_SignlFilter_ms       := _20_AUTO.recipe.st120.FeederConfigRight.InFilterDelay,
               diIN_StartDelay_ms        := _20_AUTO.recipe.st120.FeederConfigRight.StartDelay,
               diIN_StopDelay_ms         := _20_AUTO.recipe.st120.FeederConfigRight.StopDelay,
               diIN_EmptyDelay_ms        := _20_AUTO.recipe.st120.FeederConfigRight.EmptyDelay);

simu_feederLeft(xIN_Enable         := FEEDER_SIMULATION AND CONST.USE_SIMULATION,
                xIN_PceSensor      := IO_BOX.I8304_ST120_maxi_zufurung_links,
                tIN_NewPieceTime   := 500,
                iIN_WaitTimeMin_ms := 1000,
                iIN_WaitTimeMax_ms := 1500);

simu_feederRight(xIN_Enable         := FEEDER_SIMULATION AND CONST.USE_SIMULATION,
                 xIN_PceSensor      := IO_BOX.I8305_ST120_maxi_zufurung_rechts,
                 tIN_NewPieceTime   := 500,
                 iIN_WaitTimeMin_ms := 1000,
                 iIN_WaitTimeMax_ms := 1500);

fb_hubladerLeft(xIN_Reset    := xIN_Reset OR (ST120_Feeder_e.RESET = iOUT_Step),
                xIN_Quit     := xIN_Quit,
                xIN_Manu     := enState.StateMANU = enIN_State,
                pbtIN_Button := ADR(HMI.btManuCylinders[StationList_e.ST120][5]),
                xIN_GS       := simu_hubladerLeft.xOUT_inGS,
                xIN_AS       := simu_hubladerLeft.xOUT_inAS,
                xIN_FREE     := TRUE,
                xINtoGS      := fb_feederLeft.xOUT_EnableFeeder AND fb_hubladerLeft.xIN_AS,
                xINtoAS      := fb_feederLeft.xOUT_EnableFeeder AND fb_hubladerLeft.xIN_GS,
                tIN_ErrAS    := DINT_TO_TIME(_20_AUTO.recipe.cylinder2Pos[StationList_e.ST120]
                                                 [ST120_Cylinders_e.HubladerLinks].toAS_alarm_time),
                tIN_ErrGS := DINT_TO_TIME(_20_AUTO.recipe.cylinder2Pos[StationList_e.ST120]
                                              [ST120_Cylinders_e.HubladerLinks].toGS_alarm_time),
                tIN_WaitAS := DINT_TO_TIME(_20_AUTO.recipe.cylinder2Pos[StationList_e.ST120]
                                               [ST120_Cylinders_e.HubladerLinks].toAS_wait_time),
                tIN_WaitGS := DINT_TO_TIME(_20_AUTO.recipe.cylinder2Pos[StationList_e.ST120]
                                               [ST120_Cylinders_e.HubladerLinks].toGS_wait_time));

simu_hubladerLeft(xIN_Enable := FEEDER_SIMULATION AND CONST.USE_SIMULATION,
                  xIN_inGS   := IO_BOX.I8204_ST120_hublader_links_unten,
                  xIN_inAS   := IO_BOX.I8205_ST120_hublader_links_oben,
                  xIN_valve  := fb_hubladerLeft.xOUT_VALVE,
                  tIN_GS_ms  := 800,  //ms
                  tIN_AS_ms  := 800); //ms

fb_hubladerRight(xIN_Reset    := xIN_Reset OR (ST120_Feeder_e.RESET = iOUT_Step),
                 xIN_Quit     := xIN_Quit,
                 xIN_Manu     := enState.StateMANU = enIN_State,
                 pbtIN_Button := ADR(HMI.btManuCylinders[StationList_e.ST120][6]),
                 xIN_GS       := simu_hubladerRight.xOUT_inGS,
                 xIN_AS       := simu_hubladerRight.xOUT_inAS,
                 xIN_FREE     := TRUE,
                 xINtoGS      := fb_feederRight.xOUT_EnableFeeder AND fb_hubladerRight.xIN_AS,
                 xINtoAS      := fb_feederRight.xOUT_EnableFeeder AND fb_hubladerRight.xIN_GS,
                 tIN_ErrAS    := DINT_TO_TIME(_20_AUTO.recipe.cylinder2Pos[StationList_e.ST120]
                                                  [ST120_Cylinders_e.HubladerRechts].toAS_alarm_time),
                 tIN_ErrGS := DINT_TO_TIME(_20_AUTO.recipe.cylinder2Pos[StationList_e.ST120]
                                               [ST120_Cylinders_e.HubladerRechts].toGS_alarm_time),
                 tIN_WaitAS := DINT_TO_TIME(_20_AUTO.recipe.cylinder2Pos[StationList_e.ST120]
                                                [ST120_Cylinders_e.HubladerRechts].toAS_wait_time),
                 tIN_WaitGS := DINT_TO_TIME(_20_AUTO.recipe.cylinder2Pos[StationList_e.ST120]
                                                [ST120_Cylinders_e.HubladerRechts].toGS_wait_time));

simu_hubladerRight(xIN_Enable := FEEDER_SIMULATION AND CONST.USE_SIMULATION,
                   xIN_inGS   := IO_BOX.I8300_ST120_hublader_rechts_unten,
                   xIN_inAS   := IO_BOX.I8301_ST120_hublader_rechts_oben,
                   xIN_valve  := fb_hubladerRight.xOUT_VALVE,
                   tIN_GS_ms  := 800,  //ms
                   tIN_AS_ms  := 800); //ms

rtPutPieceLeft(CLK := simu_hubladerLeft.xOUT_inAS);
rtPutPieceRight(CLK := simu_hubladerRight.xOUT_inAS);

IF rtPutPieceLeft.Q THEN
    simu_fifoLeft.Put(1);
END_IF

IF rtPutPieceRight.Q THEN
    simu_fifoRight.Put(1);
END_IF

(*******************************************************************)
(* OUTPUTS *)
(*******************************************************************)
// Error Flag 
xOUT_ErrFlag := (bOUT_Error <> 0) OR (ST120_Feeder_e.ERROR = iOUT_Step);
// Baustein befindet sich im Ablauf 
xOUT_Busy := (iOUT_Step > ST120_Feeder_e.READY) AND (iOUT_Step < ST120_Feeder_e.DONE);
// Baustein hat den Ablauf beendet
xOUT_Done := (iOUT_Step = ST120_Feeder_e.DONE);
// Process ready
xOUT_Ready := (iOUT_Step = ST120_Feeder_e.READY);
// Timeout FB 				 		
xOUT_Timeout := TON_Timeout.Q;
// Itialisierung fertig			
xOUT_InitDone := (iOUT_Step = ST120_Feeder_e.READY);
// Aktueller Schritt			
iOUT_Step := iOUT_Step; //Im Ablauf gesetzt		
sOUT_Step := TO_STRING(iOUT_Step);
//Fehlernummer	 
bOUT_Error := bOUT_Error; //Im Ablauf/FB gesetzt	
(* Warte (alle Schritte wo auf FG oder Teile gewartet wird) *)
xOUT_Wait := (iOUT_Step = ST120_Feeder_e.DONE) OR
             (iOUT_Step = ST120_Feeder_e.READY);

IO_BOX.Q5204_14_ST120_schwenken_links :=
    fb_pivotLeft.xOUT_VALVE AND NOT (FEEDER_SIMULATION AND CONST.USE_SIMULATION);

IO_BOX.Q5205_14_ST120_schwenken_rechts :=
    fb_pivotRight.xOUT_VALVE AND NOT (FEEDER_SIMULATION AND CONST.USE_SIMULATION);

IO_BOX.Q8207_ST120_hublader_links_valve :=
    fb_hubladerLeft.xOUT_VALVE AND NOT (FEEDER_SIMULATION AND CONST.USE_SIMULATION);

IO_BOX.Q8303_ST120_hublader_rechts_valve :=
    fb_hubladerRight.xOUT_VALVE AND NOT (FEEDER_SIMULATION AND CONST.USE_SIMULATION);

IO_BOX.Q8201_ST120_forderband_ein_l :=
    (enIN_State = enState.StateAUTO) AND
    NOT (FEEDER_SIMULATION AND CONST.USE_SIMULATION);

IO_BOX.Q8203_ST120_forderband_ein_r :=
    (enIN_State = enState.StateAUTO) AND
    NOT (FEEDER_SIMULATION AND CONST.USE_SIMULATION);

(*******************************************************************)
(* Ablauf *)
(*******************************************************************)

(* Sperren *)
IF xIN_Sperre THEN
    iPreStep  := ST120_Feeder_e.RESET;
    iOUT_Step := ST120_Feeder_e.RESET;
    RETURN;
END_IF;

(* Schritt Merker *)
IF iAktStep <> iOUT_Step THEN
    iLastStep := iAktStep;
    iAktStep  := iOUT_Step;
END_IF

(* START *)
rtSTART(CLK := xIN_Start);

(* error management *)
IF 0 = bOUT_Error THEN
    IF fb_pivotLeft.xOUT_ErrFlag THEN
        bOUT_Error := ST120_Alarm_e.Cylinder_pivot_left;
    ELSIF fb_pivotRight.xOUT_ErrFlag THEN
        bOUT_Error := ST120_Alarm_e.Cylinder_pivot_right;
    ELSIF fb_hubladerLeft.xOUT_ErrFlag THEN
        bOUT_Error := ST120_Alarm_e.Cylinder_hublader_left;
    ELSIF fb_hubladerRight.xOUT_ErrFlag THEN
        bOUT_Error := ST120_Alarm_e.Cylinder_hublader_right;
    END_IF
ELSIF iOUT_Step < ST120_Feeder_e.ERROR THEN
    iOUT_Step := ST120_Feeder_e.ERROR;
END_IF

(*******************************************************************)
(* Schrittkette  *)
(*******************************************************************)
CASE iOUT_Step OF

(***** RESET *****)
ST120_Feeder_e.RESET: (* Schritt 0-99 *)
    //Initialisierungen
    //Start Init Ablauf
    IF xIN_Init THEN
        iOUT_Step := ST120_Feeder_e.INIT;
        //Start Manu Ablauf
    ELSIF enIN_State = StateMANU AND xIN_NextStep THEN
        iOUT_Step := ST120_Feeder_e.INIT;
    END_IF;

(***** INIT *****)
ST120_Feeder_e.INIT: (* Grundstellung ? *)
    IF xIN_PnpGripperOpen AND xIN_PnpNotOnTheWay THEN
        iOUT_Step := ST120_Feeder_e.Init_pneumatics;
    END_IF;

ST120_Feeder_e.Init_pneumatics:
    // TODO check all the sensors
    IF FEEDER_SIMULATION AND CONST.USE_SIMULATION THEN
        iOUT_Step := ST120_Feeder_e.Init_pivot_to_feeder;
    ELSE
        IF (NOT _20_AUTO.recipe.st120.xUseVerLeft AND IO_BOX.I6404_ST120_teil_in_vereizelung_links) OR
           (NOT _20_AUTO.recipe.st120.xUseVerRight AND IO_BOX.I6405_ST120_teil_in_vereinzelung_rechts) THEN
            bOUT_Error := ST120_Alarm_e.Piece_in_unused_pivot;
            iOUT_Step  := ST120_Feeder_e.ERROR;

        ELSIF (IO_BOX.I6401_ST120_schwenken_links_in_horizontal AND
               IO_BOX.I6403_ST120_schwenken_rechts_in_horizontal) THEN
            iOUT_Step := ST120_Feeder_e.Init_pivot_to_feeder;

        ELSIF (_20_AUTO.recipe.st120.xUseVerLeft AND NOT IO_BOX.I6404_ST120_teil_in_vereizelung_links) AND
              (_20_AUTO.recipe.st120.xUseVerRight AND IO_BOX.I6405_ST120_teil_in_vereinzelung_rechts) THEN
            bOUT_Error := ST120_Alarm_e.Piece_missing_left_pivot;
            iOUT_Step  := ST120_Feeder_e.ERROR;

        ELSIF (_20_AUTO.recipe.st120.xUseVerLeft AND IO_BOX.I6404_ST120_teil_in_vereizelung_links) AND
              (_20_AUTO.recipe.st120.xUseVerRight AND NOT IO_BOX.I6405_ST120_teil_in_vereinzelung_rechts) THEN
            bOUT_Error := ST120_Alarm_e.Piece_missing_right_pivor;
            iOUT_Step  := ST120_Feeder_e.ERROR;

        ELSIF NOT IO_BOX.I6404_ST120_teil_in_vereizelung_links AND NOT IO_BOX.I6405_ST120_teil_in_vereinzelung_rechts
            THEN
            iOUT_Step := ST120_Feeder_e.Init_pivot_to_feeder;

        ELSE
            iOUT_Step := ST120_Feeder_e.Init_pivot_to_pnp;
        END_IF
    END_IF

ST120_Feeder_e.Init_pivot_to_feeder:
    IF (NOT _20_AUTO.recipe.st120.xUseVerLeft OR fb_pivotLeft.xOUT_inAS) AND
       (NOT _20_AUTO.recipe.st120.xUseVerRight OR fb_pivotRight.xOUT_inAS) THEN
        iOUT_Step := ST120_Feeder_e.READY;
    END_IF

ST120_Feeder_e.Init_pivot_to_pnp:
    IF (NOT _20_AUTO.recipe.st120.xUseVerLeft OR fb_pivotLeft.xOUT_inGS) AND
       (NOT _20_AUTO.recipe.st120.xUseVerRight OR fb_pivotRight.xOUT_inGS) THEN
        iOUT_Step := ST120_Feeder_e.READY;
    END_IF

(***** READY / INIT DONE *****)
ST120_Feeder_e.READY: (* Start AUTO,END,LEER,STEP *)
    IF xIN_Start THEN //IF rtSTART.Q THEN
        iOUT_Step := ST120_Feeder_e.START;
    END_IF

(***** START  ZYKLISCH *****)
ST120_Feeder_e.START: (*  *)
    IF xIN_NextStep AND pxFG_Freigabe^ THEN
        iOUT_Step := ST120_Feeder_e.wait_tube_presence;
    END_IF;

ST120_Feeder_e.wait_tube_presence:
    IF (FEEDER_SIMULATION AND CONST.USE_SIMULATION) THEN
        IF (NOT _20_AUTO.recipe.st120.xUseVerLeft OR (simu_fifoLeft.GetLen() >= BAND_SIZE_FOR_TUBE_LEFT)) AND
           (NOT _20_AUTO.recipe.st120.xUseVerRight OR (simu_fifoRight.GetLen() >= BAND_SIZE_FOR_TUBE_RIGHT)) THEN
            iOUT_Step := ST120_Feeder_e.wait_pnp_ready;
        END_IF

    ELSE
        IF (NOT _20_AUTO.recipe.st120.xUseVerLeft OR TON_PieceInPivotLeft.Q) AND
           (NOT _20_AUTO.recipe.st120.xUseVerRight OR TON_PieceInPivotRight.Q) THEN
            iOUT_Step := ST120_Feeder_e.wait_pnp_ready;
        END_IF
    END_IF

ST120_Feeder_e.wait_pnp_ready:
    IF xIN_PnpGripperOpen THEN
        iOUT_Step := ST120_Feeder_e.rotate_to_pnp;
    END_IF

ST120_Feeder_e.rotate_to_pnp:
    IF fb_pivotLeft.xOUT_inGS AND fb_pivotRight.xOUT_inGS THEN
        iOUT_Step := ST120_Feeder_e.wait_pce_picked;
    END_IF

ST120_Feeder_e.wait_pce_picked:
    IF xIN_PickPiece THEN
        IF _20_AUTO.recipe.st120.xUseVerLeft THEN
            simu_fifoLeft.Pop(1);
        END_IF

        IF _20_AUTO.recipe.st120.xUseVerRight THEN
            simu_fifoRight.Pop(1);
        END_IF

        iOUT_Step := ST120_Feeder_e.wait_pnp_move_out_with_the_piece;
    END_IF

ST120_Feeder_e.wait_pnp_move_out_with_the_piece:
    IF xIN_PnpNotOnTheWay THEN
        iOUT_Step := ST120_Feeder_e.rotate_to_feeder;
    END_IF

ST120_Feeder_e.rotate_to_feeder:
    IF (NOT _20_AUTO.recipe.st120.xUseVerLeft OR fb_pivotLeft.xOUT_inAS) AND
       (NOT _20_AUTO.recipe.st120.xUseVerRight OR fb_pivotRight.xOUT_inAS) THEN
        iOUT_Step := ST120_Feeder_e.DONE;
    END_IF

(***** DONE *****)
ST120_Feeder_e.DONE: (* Letzter Schritt  *)
    IF NOT xIN_AlarmAktiv THEN
        //AUTO
        IF (enIN_State = StateAUTO) AND xIN_RestartCYCL THEN
            iOUT_Step := ST120_Feeder_e.START;
            //STEP / END / LEERFAHREN restart
        ELSIF (enIN_State < StateAUTO) AND (enIN_State >= enState.StateSTEP) AND xIN_RestartCYCL THEN
            iOUT_Step := ST120_Feeder_e.START;
            //STEP / END / LEERFAHREN fertig
        ELSIF (enIN_State = StateREADY) THEN
            iOUT_Step := ST120_Feeder_e.READY;
        END_IF;
    END_IF;

(************ ERROR *************)
ST120_Feeder_e.ERROR: (* ERROR *) ;

END_CASE;

END_FUNCTION_BLOCK

// ---- POUs/20_AUTO/ST125/FB_AUT_125.TcPOU
FUNCTION_BLOCK FB_AUT_125 EXTENDS FB_AUT_ABSTRACT
(****************************************************************************)
(*	POU_AUT_zxx			Bausteinaufrufe Station	zxx							*)
(*	Status				ungetestet											*)
(*  Version:			1.0													*)
(*	Beschrieb:																*)
(*																			*)
(*	Abläufe:			FB_ABLzxxA		Hauptablauf							*)
(*																			*)
(*																			*)
(* 	25.09.2019/Dj															*)
(****************************************************************************)
(*	dd.mm.yyyy   KZ    x.y			Beschrieb								*)
(****************************************************************************)
VAR_INPUT
    (* spezifische Eingänge *)

END_VAR
VAR_OUTPUT
    (* spezifische Ausgänge *)

END_VAR
VAR
    (* Bausteine *)
    fb_Pnp    : FB_ABL_125_Pnp;
    fb_Feeder : FB_ABL_125_Feeder;

    fb_stat_pnp    : FB_AUT_Statistics;
    fb_stat_Feeder : FB_AUT_Statistics;

END_VAR

VAR CONSTANT
    ROT_TABLE_FREE_MAX_Y : REAL := 200.0; // If Y and Z axis is more than this value, the feeder cannot move
    ROT_TABLE_FREE_MAX_Z : REAL := 200.0; // If Z and Y axis is more than this value, the feeder cannot move
END_VAR

(*******************************************************************)
(* Timer *)
(*******************************************************************)

(*******************************************************************)
(* Flanken / Merker *)
(*******************************************************************)
//MANU CYCLE
IF (enIN_State = StateMANU) AND xIN_ManuCycle THEN
    xManuCycle := TRUE;
END_IF;

IF (enIN_State <> StateMANU) OR xOUT_Done THEN
    xManuCycle := FALSE;
END_IF

//NEXT STEP
xNextStep := (enIN_State > StateSTEP) OR
             ((enIN_State = StateSTEP) AND xIN_Step) OR
             ((enIN_State = StateMANU) AND xManuCycle);

//RESET
xReset := (enIN_State < StateREADY) AND (enIN_State <> StateINIT) AND NOT xManuCycle;

(*******************************************************************)
(* Bausteinaufrufe Abläufe *)
(*******************************************************************)

xRelease := MAIN.MoverMan.IsProcessUsed(THIS^);

fb_Pnp(xIN_Reset          := xReset,
       xIN_Init           := xIN_Init,
       xIN_Quit           := xIN_Quit,
       xIN_Start          := enIN_State >= enState.StateLEER AND xRelease,
       xIN_Sperre         := NOT xIN_On,
       xIN_NextStep       := xNextStep,
       xIN_AlarmAktiv     := xIN_AlarmAktiv,
       xIN_DryCycle       := xIN_DryCycle,
       xIN_RestartCYCL    := enIN_State >= enState.StateLEER,
       enIN_State         := enIN_State,
       tIN_Timeout        := tIN_Timeout,
       pxFG_Freigabe      := ADR(xRelease),
       Mover              := THIS^.Mover,
       xIN_PceReadyToPick := fb_Feeder.xOUT_Done);

fb_Feeder(xIN_Reset       := xReset,
          xIN_Init        := xIN_Init,
          xIN_Quit        := xIN_Quit,
          xIN_Start       := enIN_State >= enState.StateLEER AND xRelease,
          xIN_Sperre      := NOT xIN_On,
          xIN_NextStep    := xNextStep,
          xIN_AlarmAktiv  := xIN_AlarmAktiv,
          xIN_DryCycle    := xIN_DryCycle,
          xIN_RestartCYCL := enIN_State >= enState.StateLEER,
          enIN_State      := enIN_State,
          tIN_Timeout     := tIN_Timeout,
          pxFG_Freigabe   := ADR(xRelease),
          // special
          xIN_PickPiece            := fb_Pnp.xOUT_PickPiece,
          xIN_RotTableBlockedByPnp := (ST125_Axis.axis125_01Y.rActPos > ROT_TABLE_FREE_MAX_Y) AND
                                      (ST125_Axis.axis125_02Z.rActPos > ROT_TABLE_FREE_MAX_Z));

fb_stat_pnp(xIN_Enable  := enState.StateAUTO = enIN_State,
            xIN_Waiting := fb_Pnp.xOUT_Wait,
            xIN_Running := (fb_Pnp.iOUT_Step >= ST125_Pnp_e.START) AND
                           (fb_Pnp.iOUT_Step <= ST125_Pnp_e.DONE),
            // Since we use a mover system, a cycle is done when we are waiting on a mover
            xIN_Done := fb_Pnp.iOUT_Step = ST125_Pnp_e.waitOnMover);

fb_stat_Feeder(xIN_Enable  := enState.StateAUTO = enIN_State,
               xIN_Waiting := fb_feeder.xOUT_Wait,
               xIN_Running := (fb_feeder.iOUT_Step >= ST125_Feeder_e.START) AND
                              (fb_feeder.iOUT_Step <= ST125_Feeder_e.DONE),
               xIN_Done := fb_feeder.iOUT_Step = ST125_Feeder_e.DONE);

(*******************************************************************)
(* Mover reset flags *)
(*******************************************************************)

(*******************************************************************)
(* OUTPUT *)
(*******************************************************************)
xOUT_InitDone := fb_Pnp.xOUT_InitDone AND fb_Feeder.xOUT_InitDone;
xOUT_Ready    := fb_Pnp.xOUT_Ready AND fb_Feeder.xOUT_Ready;
xOUT_Done     := fb_Pnp.xOUT_Done;
xOUT_ErrFlag  := fb_Pnp.xOUT_ErrFlag OR fb_Feeder.xOUT_ErrFlag;
xOUT_Wait     := fb_Pnp.xOUT_Wait AND fb_Feeder.xOUT_Wait;
xOUT_AlarmST  := xOUT_ErrFlag;

IF fb_Pnp.xOUT_ErrFlag THEN
    bOUT_ErrorNum := fb_Pnp.bOUT_Error;
ELSIF fb_Feeder.xOUT_ErrFlag THEN
    bOUT_ErrorNum := fb_Feeder.bOUT_Error;
ELSE
    bOUT_ErrorNum := 0;
END_IF

(*******************************************************************)
(* Bausteinaufruf Error Station *)
(*******************************************************************)
POU_ALARM_125(xIN_QUIT      := xIN_Quit,
              iIN_ArraySize := ST125_Alarm_e._max,
              pstrIN_ALARM  := ADR(HMI.strArALARM[81]),
              refPOU        := THIS^);

(* % of completion of the process *)
PROPERTY iCompletionPC : INT
GET
iCompletionPC := THIS^.fb_Pnp.iOUT_ProcessCompletion;
END_GET
END_PROPERTY

PROPERTY ProcessExecution : ProcessExecution_e
GET
ProcessExecution := THIS^._ProcessExecution;
END_GET
SET
THIS^._ProcessExecution := ProcessExecution;
END_SET
END_PROPERTY

PROPERTY xBusy : BOOL
GET
xBusy := THIS^.fb_Pnp.xOUT_Busy;
END_GET
SET
END_SET
END_PROPERTY

PROPERTY xDone : BOOL
GET
xDone := THIS^.fb_Pnp.xOUT_Ready OR THIS^.fb_Pnp.xOUT_Done;
END_GET
END_PROPERTY

PROPERTY xMoverPathFree : BOOL
GET
xMoverPathFree := THIS^.fb_Pnp.xOUT_MoverFree OR THIS^.fb_Pnp.xOUT_Ready OR THIS^.fb_Pnp.xOUT_Done;
END_GET
END_PROPERTY

PROPERTY xMoverShouldLeave : BOOL
GET
xMoverShouldLeave := THIS^.fb_Pnp.iOUT_Step = ST125_Pnp_e.SYNC_MOVER_LEAVE;
END_GET
END_PROPERTY

END_FUNCTION_BLOCK

// ---- POUs/20_AUTO/ST125/FB_ABL_125_Pnp.TcPOU
FUNCTION_BLOCK FB_ABL_125_Pnp
(****************************************************************************************)
(*	TITEL				laden kristall- Modul	    										*)
(*	Status				ungetestet                         								*)
(*	Beschrieb:			Ablaufbeschreibung												*)
(*																						*)
(*	Steps:	self-explained using enum													*)
(***********************************Revisionen*******************************************)
(*	see github blames																	*)
(****************************************************************************************)

VAR_INPUT
    xIN_Reset       : BOOL;          // Schrittkette zurücksetzen 
    xIN_Init        : BOOL;          // Initialisieren
    xIN_Quit        : BOOL;          // Fehler quittieren 
    xIN_Start       : BOOL;          // Startbefehl
    xIN_Sperre      : BOOL;          // FB Sperren 
    xIN_NextStep    : BOOL;          // Nächsten Schritt ausführen 
    xIN_AlarmAktiv  : BOOL;          // Anlage hat Alarm
    xIN_DryCycle    : BOOL;          // Fahren ohne Teile
    xIN_RestartCYCL : BOOL;          // Zyklus erneut starten im STEP, END, LEERFAHREN
    enIN_State      : enState;       // Status Anlage
    tIN_Timeout     : TIME := T#10s; // Timout

    pxFG_Freigabe : POINTER TO BOOL; //Freigabe von Station

    // Application specific
    Mover              : REFERENCE TO FB_Mover;
    xIN_PceReadyToPick : BOOL; // the piece(s) is/are ready to picked
END_VAR
VAR_OUTPUT
    (* standart Ausgänge *)
    xOUT_ErrFlag  : BOOL;        // Error Flag 
    xOUT_Busy     : BOOL;        // Baustein befindet sich im Ablauf 
    xOUT_Done     : BOOL;        // Baustein hat den Ablauf beendet 		
    xOUT_Ready    : BOOL;        // Ready to begin, should be the same state as done	
    xOUT_Timeout  : BOOL;        // Timeout FB 
    xOUT_InitDone : BOOL;        // initialisierung fertig
    xOUT_Wait     : BOOL;        // Wartet auf Bedingung
    iOUT_Step     : ST125_Pnp_e; // Aktueller Schritt 
    sOUT_Step     : STRING;      // Aktueller Schritt but in string format
    bOUT_Error    : BYTE;        // Fehlernummer

    iOUT_ProcessCompletion : INT;  //process completion, express in % (0-100)
    xOUT_MoverFree         : BOOL; // The mover is free to move
    xOUT_PickPiece         : BOOL; // Set to true when a piece is picked

END_VAR
VAR
    (* Standard *)
    (* Schritt *)
    iLastStep : ST125_Pnp_e; // Merker letzter Schritt 
    iPreStep  : ST125_Pnp_e; // Schritt zurück nach Alarm 
    iAktStep  : ST125_Pnp_e; // aktueller Schritt

    // Trigger Starten 
    rtSTART : R_TRIG;
    // Timer TimeOut 
    TON_Timeout : TON;

    (* Bausteine *)

    (* Spezial *)
    fb_axis125_01Y : FB_AxisLM_V1_1;
    fb_axis125_02Z : FB_AxisLM_V1_1;

    fb_PnpHorAxis : FB_LinearMotionMan;
    fb_PnpVerAxis : FB_LinearMotionMan;

    fb_simu_axis125_01Y : FB_Simu_AxisLM_V1_1;
    fb_simu_axis125_02Z : FB_Simu_AxisLM_V1_1;

    fb_gripperFilterhutLeft    : FB_ZylMo2El_V2_1;
    fb_gripperFilterhutRight   : FB_ZylMo2El_V2_1;
    simu_gripperFilterhutLeft  : FB_Simu_Zyl2Pos;
    simu_gripperFilterhutRight : FB_Simu_Zyl2Pos;

    fb_handlingSolerohrLeft    : FB_ZylMo2El_V2_1;
    fb_handlingSolerohrRight   : FB_ZylMo2El_V2_1;
    simu_handlingSolerohrLeft  : FB_Simu_Zyl2Pos;
    simu_handlingSolerohrRight : FB_Simu_Zyl2Pos;

    fb_gripperSolerohrLeft    : FB_ZylMo2El_V2_1;
    fb_gripperSolerohrRight   : FB_ZylMo2El_V2_1;
    simu_gripperSolerohrLeft  : FB_Simu_Zyl2Pos;
    simu_gripperSolerohrRight : FB_Simu_Zyl2Pos;

    fb_kraftLeft  : FB_WandlerForceSensor;
    fb_kraftRight : FB_WandlerForceSensor;

END_VAR
VAR CONSTANT
    PNP_SIMULATION       : BOOL := FALSE; // Set to TRUE to simulate this part of the program
    PNP_DONT_CHECK_KRAFT : BOOL := FALSE; // set to TRUE if you won't check kraft
END_VAR

(*******************************************************************)
(* Trigger  *)
(*******************************************************************)
(* Zurücksetzen *)
IF xIN_RESET THEN
    iPreStep  := ST125_Pnp_e.RESET;
    iOUT_Step := ST125_Pnp_e.RESET;
END_IF;

(* Error Quittieren *)
IF (bOUT_Error <> 0) AND xIN_Quit THEN
    xOUT_ErrFlag := FALSE;
    bOUT_Error   := 0;
    iOUT_Step    := iPreStep;
END_IF;

(*******************************************************************)
(* Timer *)
(*******************************************************************)
TON_Timeout(IN := xIN_NextStep AND (iLastStep = iOUT_Step) (*todo FG *) ,
            PT := tIN_Timeout);

(*******************************************************************)
(* Bausteine *)
(*******************************************************************)
fb_PnpHorAxis(config          := _20_AUTO.recipe.linearAxis[LinearAxis_e.ST125_01Y],
              xIN_Init        := enIN_State = enState.StateINIT,
              xIN_Reset       := xIN_Reset,
              lrIN_CurrPos    := fb_axis125_01Y.rOUT_ActPos,
              lrIN_Delta_mm   := 0.5,
              iIN_CurrentStep := iOUT_Step,
              iIN_moveNumber  := ST125_PnpHorPos_e._max);

fb_simu_axis125_01Y(xIN_Enable          := PNP_SIMULATION AND CONST.USE_SIMULATION,
                    bIN_AxisCntr        := fb_axis125_01Y.bOUT_AxisCntr,
                    wIN_AxisState       := ST125_Axis.axis125_01Y.wState,
                    udiIN_HomingTime_ms := 2000,
                    pIN_axisSimu        := ADR(SIMU.axis_ref[Axis_e.ST125_01Y]),
                    pIN_axisHW          := ADR(ST125_Axis.axis125_01Y.axis),
                    rIN_PosActual       := fb_axis125_01Y.rOUT_ActPos,
                    rIN_PosMax          := ST125_Axis.const125_01Y.POS_MAX,
                    rIN_PosMin          := ST125_Axis.const125_01Y.POS_MIN,
                    rIN_PixMax          := 100,
                    rIN_PixMin          := 0);

fb_axis125_01Y(enIN_State       := enIN_State,
               parIN_Buttons    := ADR(AXIS.btTeachArAxis[Axis_e.ST125_01Y]),
               xIN_DisButtons   :=,
               xIN_Quit         := xIN_Quit,
               xIN_PARAMok      := TRUE, (*TODO*)
               xIN_FREE         := TRUE,
               xIN_FREE_HOME    := TRUE,
               rIN_POSMIN       := ST125_Axis.const125_01Y.POS_MIN,
               rIN_POSMAX       := ST125_Axis.const125_01Y.POS_MAX,
               rIN_VELOMAX      := ST125_Axis.const125_01Y.VELO_MAX,
               rIN_VELOMANU     := ST125_Axis.const125_01Y.VELO_MANU,
               rIN_VELOOPEN     := ST125_Axis.const125_01Y.VELO_MANU / 4,
               rIN_JogInc       := AXIS.rTeachIncAxis,
               xIN_Execute      := fb_PnpHorAxis.xOUT_Execute,
               xIN_Home         := ST125_Pnp_e.Init_HomeHorizontals = iAktStep,
               xIN_Relative     :=,
               rIN_Position     := TO_REAL(fb_PnpHorAxis.OUT_MoveProfile.lrPosition),
               rIN_Velocity     := TO_REAL(fb_PnpHorAxis.OUT_MoveProfile.lrVelocity),
               rIN_Acceleration := TO_REAL(fb_PnpHorAxis.OUT_MoveProfile.lrAccel),
               rIN_Deceleration := TO_REAL(fb_PnpHorAxis.OUT_MoveProfile.lrDecel),
               rIN_Jerk         := TO_REAL(fb_PnpHorAxis.OUT_MoveProfile.lrJerk),
               rIN_PosManu      :=
               TO_REAL(_20_AUTO.recipe
                           .linearAxis[LinearAxis_e.ST125_01Y].movesList[AXIS.bTeachPos[Axis_e.ST125_01Y]].lrPosition),
               rIN_VeloJogManu := TO_REAL(Axis.rJogVelo_pc),
               xIN_Reset       := (ST125_Pnp_e.RESET = iAktStep) OR xIN_Reset,
               // the simu fb gives the hardware signal when the simulation is disabled
               wAxisState    := fb_simu_axis125_01Y.wOUT_AxisState,
               bOUT_AxisCntr => ST125_Axis.axis125_01Y.bCtrlHi,
               rOUT_ActPos   => ST125_Axis.axis125_01Y.rActPos,
               axisIN_REF    := fb_simu_axis125_01Y.pOUT_axisRef^);

fb_PnpVerAxis(config          := _20_AUTO.recipe.linearAxis[LinearAxis_e.ST125_02Z],
              xIN_Init        := enIN_State = enState.StateINIT,
              xIN_Reset       := xIN_Reset,
              lrIN_CurrPos    := fb_axis125_02Z.rOUT_ActPos,
              lrIN_Delta_mm   := 0.5,
              iIN_CurrentStep := iOUT_Step,
              iIN_moveNumber  := ST125_PnpVerPos_e._max);

fb_simu_axis125_02Z(xIN_Enable          := PNP_SIMULATION AND CONST.USE_SIMULATION,
                    bIN_AxisCntr        := fb_axis125_02Z.bOUT_AxisCntr,
                    wIN_AxisState       := ST125_Axis.axis125_02Z.wState,
                    udiIN_HomingTime_ms := 2000,
                    pIN_axisSimu        := ADR(SIMU.axis_ref[Axis_e.ST125_02Z]),
                    pIN_axisHW          := ADR(ST125_Axis.axis125_02Z.axis),
                    rIN_PosActual       := fb_axis125_02Z.rOUT_ActPos,
                    rIN_PosMax          := ST125_Axis.const125_02Z.POS_MAX,
                    rIN_PosMin          := ST125_Axis.const125_02Z.POS_MIN,
                    rIN_PixMax          := 80,
                    rIN_PixMin          := 0);

fb_axis125_02Z(enIN_State       := enIN_State,
               parIN_Buttons    := ADR(AXIS.btTeachArAxis[Axis_e.ST125_02Z]),
               xIN_DisButtons   :=,
               xIN_Quit         := xIN_Quit,
               xIN_PARAMok      := TRUE, (*TODO*)
               xIN_FREE         := TRUE,
               xIN_STOP         := (iOUT_Step = ST125_Pnp_e.PnP_Ver_quick_stop),
               xIN_FREE_HOME    := TRUE,
               rIN_POSMIN       := ST125_Axis.const125_02Z.POS_MIN,
               rIN_POSMAX       := ST125_Axis.const125_02Z.POS_MAX,
               rIN_VELOMAX      := ST125_Axis.const125_02Z.VELO_MAX,
               rIN_VELOMANU     := ST125_Axis.const125_02Z.VELO_MANU,
               rIN_VELOOPEN     := ST125_Axis.const125_02Z.VELO_MANU / 4,
               rIN_JogInc       := AXIS.rTeachIncAxis,
               xIN_Execute      := fb_PnpVerAxis.xOUT_Execute,
               xIN_Home         := ST125_Pnp_e.Init_HomeVerticals = iAktStep,
               xIN_Relative     :=,
               rIN_Position     := TO_REAL(fb_PnpVerAxis.OUT_MoveProfile.lrPosition),
               rIN_Velocity     := TO_REAL(fb_PnpVerAxis.OUT_MoveProfile.lrVelocity),
               rIN_Acceleration := TO_REAL(fb_PnpVerAxis.OUT_MoveProfile.lrAccel),
               rIN_Deceleration := TO_REAL(fb_PnpVerAxis.OUT_MoveProfile.lrDecel),
               rIN_Jerk         := TO_REAL(fb_PnpVerAxis.OUT_MoveProfile.lrJerk),
               rIN_PosManu      :=
               TO_REAL(_20_AUTO.recipe
                           .linearAxis[LinearAxis_e.ST125_02Z].movesList[AXIS.bTeachPos[Axis_e.ST125_02Z]].lrPosition),
               rIN_VeloJogManu := TO_REAL(Axis.rJogVelo_pc),
               xIN_Reset       := (ST125_Pnp_e.RESET = iAktStep) OR xIN_Reset,
               // the simu fb gives the hardware signal when the simulation is disabled
               wAxisState    := fb_simu_axis125_02Z.wOUT_AxisState,
               bOUT_AxisCntr => ST125_Axis.axis125_02Z.bCtrlHi,
               rOUT_ActPos   => ST125_Axis.axis125_02Z.rActPos,
               axisIN_REF    := fb_simu_axis125_02Z.pOUT_axisRef^);

//////////////////////////////////
fb_gripperFilterhutLeft(xIN_Reset    := xIN_Reset OR (ST125_Pnp_e.RESET = iOUT_Step),
                        xIN_Quit     := xIN_Quit,
                        xIN_Manu     := enState.StateMANU = enIN_State,
                        pbtIN_Button := ADR(HMI.btManuCylinders[StationList_e.ST125][1]),
                        xIN_GS       := simu_gripperFilterhutLeft.xOUT_inGS,
                        xIN_AS       := simu_gripperFilterhutLeft.xOUT_inAS,
                        xIN_FREE     := TRUE,
                        xINtoGS      := ST125_Pnp_e.Pnp_takeTubeCap = iOUT_Step,
                        xINtoAS      := (ST125_Pnp_e.Pnp_placeCap = iOUT_Step) OR
                                        (ST125_Pnp_e.Init_open_left_clamp = iOUT_Step),
                        tIN_ErrAS := DINT_TO_TIME(_20_AUTO.recipe.cylinder2Pos[StationList_e.ST125]
                                                      [ST125_Cylinders_e.GreiferFilterhutLinks].toAS_alarm_time),
                        tIN_ErrGS := DINT_TO_TIME(_20_AUTO.recipe.cylinder2Pos[StationList_e.ST125]
                                                      [ST125_Cylinders_e.GreiferFilterhutLinks].toGS_alarm_time),
                        tIN_WaitAS := DINT_TO_TIME(_20_AUTO.recipe.cylinder2Pos[StationList_e.ST125]
                                                       [ST125_Cylinders_e.GreiferFilterhutLinks].toAS_wait_time),
                        tIN_WaitGS := DINT_TO_TIME(_20_AUTO.recipe.cylinder2Pos[StationList_e.ST125]
                                                       [ST125_Cylinders_e.GreiferFilterhutLinks].toGS_wait_time));

simu_gripperFilterhutLeft(xIN_Enable := PNP_SIMULATION AND CONST.USE_SIMULATION,
                          xIN_inGS   := IO_BOX.I6500_ST125_greiffer_filterhut_links_geschlossen,
                          xIN_inAS   := IO_BOX.I6501_ST125_greiffer_filterhut_links_offen,
                          xIN_valve  := fb_gripperFilterhutLeft.xOUT_VALVE,
                          tIN_GS_ms  := 200,  //ms
                          tIN_AS_ms  := 200); //ms

fb_gripperFilterhutRight(xIN_Reset    := xIN_Reset OR (ST125_Pnp_e.RESET = iOUT_Step),
                         xIN_Quit     := xIN_Quit,
                         xIN_Manu     := enState.StateMANU = enIN_State,
                         pbtIN_Button := ADR(HMI.btManuCylinders[StationList_e.ST125][2]),
                         xIN_GS       := simu_gripperFilterhutRight.xOUT_inGS,
                         xIN_AS       := simu_gripperFilterhutRight.xOUT_inAS,
                         xIN_FREE     := TRUE,
                         xINtoGS      := ST125_Pnp_e.Pnp_takeTubeCap = iOUT_Step,
                         xINtoAS      := ST125_Pnp_e.Pnp_placeCap = iOUT_Step OR
                                         ST125_Pnp_e.Init_open_right_clamp = iOUT_Step,
                         tIN_ErrAS := DINT_TO_TIME(_20_AUTO.recipe.cylinder2Pos[StationList_e.ST125]
                                                       [ST125_Cylinders_e.GreiferFilterhutRechts].toAS_alarm_time),
                         tIN_ErrGS := DINT_TO_TIME(_20_AUTO.recipe.cylinder2Pos[StationList_e.ST125]
                                                       [ST125_Cylinders_e.GreiferFilterhutRechts].toGS_alarm_time),
                         tIN_WaitAS := DINT_TO_TIME(_20_AUTO.recipe.cylinder2Pos[StationList_e.ST125]
                                                        [ST125_Cylinders_e.GreiferFilterhutRechts].toAS_wait_time),
                         tIN_WaitGS := DINT_TO_TIME(_20_AUTO.recipe.cylinder2Pos[StationList_e.ST125]
                                                        [ST125_Cylinders_e.GreiferFilterhutRechts].toGS_wait_time));

simu_gripperFilterhutRight(xIN_Enable := PNP_SIMULATION AND CONST.USE_SIMULATION,
                           xIN_inGS   := IO_BOX.I6502_ST125_greiffer_filterhut_rechts_geschlossen,
                           xIN_inAS   := IO_BOX.I6503_ST125_greiffer_filterhut_rechts_offen,
                           xIN_valve  := fb_gripperFilterhutRight.xOUT_VALVE,
                           tIN_GS_ms  := 200,  //ms
                           tIN_AS_ms  := 200); //ms

fb_handlingSolerohrLeft(xIN_Reset    := xIN_Reset OR (ST125_Pnp_e.RESET = iOUT_Step),
                        xIN_Quit     := xIN_Quit,
                        xIN_Manu     := enState.StateMANU = enIN_State,
                        pbtIN_Button := ADR(HMI.btManuCylinders[StationList_e.ST125][3]),
                        xIN_GS       := simu_handlingSolerohrLeft.xOUT_inGS, // TODO use sensor
                        xIN_AS       := simu_handlingSolerohrLeft.xOUT_inAS, // TODO use sensor
                        xIN_FREE     := TRUE,
                        xINtoGS      := ST125_Pnp_e.Pnp_HandlingUp = iOUT_Step OR
                                        ST125_Pnp_e.Init_handling_up = iOUT_Step,
                        // should always go down, even if this side is not used, If not, it crashes with the gripper
                        xINtoAS   := ST125_Pnp_e.Pnp_HandlingDown = iOUT_Step,
                        tIN_ErrAS := DINT_TO_TIME(_20_AUTO.recipe.cylinder2Pos[StationList_e.ST125]
                                                      [ST125_Cylinders_e.HandlingSolerohrLinks].toAS_alarm_time),
                        tIN_ErrGS := DINT_TO_TIME(_20_AUTO.recipe.cylinder2Pos[StationList_e.ST125]
                                                      [ST125_Cylinders_e.HandlingSolerohrLinks].toGS_alarm_time),
                        tIN_WaitAS := DINT_TO_TIME(_20_AUTO.recipe.cylinder2Pos[StationList_e.ST125]
                                                       [ST125_Cylinders_e.HandlingSolerohrLinks].toAS_wait_time),
                        tIN_WaitGS := DINT_TO_TIME(_20_AUTO.recipe.cylinder2Pos[StationList_e.ST125]
                                                       [ST125_Cylinders_e.HandlingSolerohrLinks].toGS_wait_time));

simu_handlingSolerohrLeft(xIN_Enable := PNP_SIMULATION AND CONST.USE_SIMULATION,
                          xIN_inGS   := IO_BOX.I6601_ST125_solerhor_handling_links_oben,
                          xIN_inAS   := IO_BOX.I6600_ST125_solerhor_handling_links_unten,
                          xIN_valve  := fb_handlingSolerohrLeft.xOUT_VALVE,
                          tIN_GS_ms  := 500,  //ms
                          tIN_AS_ms  := 500); //ms

fb_handlingSolerohrRight(xIN_Reset    := xIN_Reset OR (ST125_Pnp_e.RESET = iOUT_Step),
                         xIN_Quit     := xIN_Quit,
                         xIN_Manu     := enState.StateMANU = enIN_State,
                         pbtIN_Button := ADR(HMI.btManuCylinders[StationList_e.ST125][4]),
                         xIN_GS       := simu_handlingSolerohrRight.xOUT_inGS,
                         xIN_AS       := simu_handlingSolerohrRight.xOUT_inAS,
                         xIN_FREE     := TRUE,
                         xINtoGS      := ST125_Pnp_e.Pnp_HandlingUp = iOUT_Step OR
                                         ST125_Pnp_e.Init_handling_up = iOUT_Step,
                         // should always go down, even if this side is not used, If not, it crashes with the gripper
                         xINtoAS   := ST125_Pnp_e.Pnp_HandlingDown = iOUT_Step,
                         tIN_ErrAS := DINT_TO_TIME(_20_AUTO.recipe.cylinder2Pos[StationList_e.ST125]
                                                       [ST125_Cylinders_e.HandlingSolerohrRechts].toAS_alarm_time),
                         tIN_ErrGS := DINT_TO_TIME(_20_AUTO.recipe.cylinder2Pos[StationList_e.ST125]
                                                       [ST125_Cylinders_e.HandlingSolerohrRechts].toGS_alarm_time),
                         tIN_WaitAS := DINT_TO_TIME(_20_AUTO.recipe.cylinder2Pos[StationList_e.ST125]
                                                        [ST125_Cylinders_e.HandlingSolerohrRechts].toAS_wait_time),
                         tIN_WaitGS := DINT_TO_TIME(_20_AUTO.recipe.cylinder2Pos[StationList_e.ST125]
                                                        [ST125_Cylinders_e.HandlingSolerohrRechts].toGS_wait_time));

simu_handlingSolerohrRight(xIN_Enable := PNP_SIMULATION AND CONST.USE_SIMULATION,
                           xIN_inGS   := IO_BOX.I6603_ST125_solerhor_handling_rechts_oben,
                           xIN_inAS   := IO_BOX.I6602_ST125_solerhor_handling_rechts_unten,
                           xIN_valve  := fb_handlingSolerohrRight.xOUT_VALVE,
                           tIN_GS_ms  := 500,  //ms
                           tIN_AS_ms  := 500); //ms

fb_gripperSolerohrLeft(xIN_Reset    := xIN_Reset OR (ST125_Pnp_e.RESET = iOUT_Step),
                       xIN_Quit     := xIN_Quit,
                       xIN_Manu     := enState.StateMANU = enIN_State,
                       pbtIN_Button := ADR(HMI.btManuCylinders[StationList_e.ST125][5]),
                       xIN_GS       := simu_gripperSolerohrLeft.xOUT_inGS, // TODO use sensor
                       xIN_AS       := simu_gripperSolerohrLeft.xOUT_inAS, // TODO use sensor
                       xIN_FREE     := TRUE,
                       xINtoGS      := (ST125_Pnp_e.Pnp_HandlingSolerohrRelease = iOUT_Step) OR
                                       (ST125_Pnp_e.Init_open_solenohr_gripper = iOUT_Step),
                       xINtoAS := _20_AUTO.recipe.st125.xUseVerLeft AND
                                  (ST125_Pnp_e.Pnp_closeTubeGriper = iOUT_Step OR
                                  ST125_Pnp_e.Pnp_Ver_pushCapTorqueControl = iOUT_Step) AND
                                  fb_handlingSolerohrLeft.xOUT_inAS,
                       tIN_ErrAS := DINT_TO_TIME(_20_AUTO.recipe.cylinder2Pos[StationList_e.ST125]
                                                     [ST125_Cylinders_e.GreiferSolerohrLinks].toAS_alarm_time),
                       tIN_ErrGS := DINT_TO_TIME(_20_AUTO.recipe.cylinder2Pos[StationList_e.ST125]
                                                     [ST125_Cylinders_e.GreiferSolerohrLinks].toGS_alarm_time),
                       tIN_WaitAS := DINT_TO_TIME(_20_AUTO.recipe.cylinder2Pos[StationList_e.ST125]
                                                      [ST125_Cylinders_e.GreiferSolerohrLinks].toAS_wait_time),
                       tIN_WaitGS := DINT_TO_TIME(_20_AUTO.recipe.cylinder2Pos[StationList_e.ST125]
                                                      [ST125_Cylinders_e.GreiferSolerohrLinks].toGS_wait_time));

simu_gripperSolerohrLeft(xIN_Enable := PNP_SIMULATION AND CONST.USE_SIMULATION,
                         xIN_inGS   := IO_BOX.I6605_ST125_greifer_solerohr_links_offen,
                         // Usually you will use the sensor value, but we have too much dispersion of the pieces
                         // so it is impossible to use the sensor correctly with all kind of pices
                         // xIN_inAS   := IO_BOX.I6604_ST125_greifer_solerohr_links_geschlossen,
                         xIN_inAS  := NOT IO_BOX.I6605_ST125_greifer_solerohr_links_offen,
                         xIN_valve := fb_gripperSolerohrLeft.xOUT_VALVE,
                         tIN_GS_ms := 300,  //ms
                         tIN_AS_ms := 300); //ms

fb_gripperSolerohrRight(xIN_Reset    := xIN_Reset OR (ST125_Pnp_e.RESET = iOUT_Step),
                        xIN_Quit     := xIN_Quit,
                        xIN_Manu     := enState.StateMANU = enIN_State,
                        pbtIN_Button := ADR(HMI.btManuCylinders[StationList_e.ST125][6]),
                        xIN_GS       := simu_gripperSolerohrRight.xOUT_inGS,
                        xIN_AS       := simu_gripperSolerohrRight.xOUT_inAS,
                        xIN_FREE     := TRUE,
                        xINtoGS      := (ST125_Pnp_e.Pnp_HandlingSolerohrRelease = iOUT_Step) OR
                                        (ST125_Pnp_e.Init_open_solenohr_gripper = iOUT_Step),
                        xINtoAS := _20_AUTO.recipe.st125.xUseVerRight AND
                                   (ST125_Pnp_e.Pnp_closeTubeGriper = iOUT_Step OR
                                   ST125_Pnp_e.Pnp_Ver_pushCapTorqueControl = iOUT_Step) AND
                                   fb_handlingSolerohrRight.xOUT_inAS,
                        tIN_ErrAS := DINT_TO_TIME(_20_AUTO.recipe.cylinder2Pos[StationList_e.ST125]
                                                      [ST125_Cylinders_e.GreiferSolerohrRechts].toAS_alarm_time),
                        tIN_ErrGS := DINT_TO_TIME(_20_AUTO.recipe.cylinder2Pos[StationList_e.ST125]
                                                      [ST125_Cylinders_e.GreiferSolerohrRechts].toGS_alarm_time),
                        tIN_WaitAS := DINT_TO_TIME(_20_AUTO.recipe.cylinder2Pos[StationList_e.ST125]
                                                       [ST125_Cylinders_e.GreiferSolerohrRechts].toAS_wait_time),
                        tIN_WaitGS := DINT_TO_TIME(_20_AUTO.recipe.cylinder2Pos[StationList_e.ST125]
                                                       [ST125_Cylinders_e.GreiferSolerohrRechts].toGS_wait_time));

simu_gripperSolerohrRight(xIN_Enable := PNP_SIMULATION AND CONST.USE_SIMULATION,
                          xIN_inGS   := IO_BOX.I6607_ST125_greifer_solerohr_rechts_offen,
                          // Usually you will use the sensor value, but we have too much dispersion of the pieces
                          // so it is impossible to use the sensor correctly with all kind of pices
                          // xIN_inAS   := IO_BOX.I6606_ST125_greifer_solerohr_rechts_geschlossen,
                          xIN_inAS  := NOT IO_BOX.I6607_ST125_greifer_solerohr_rechts_offen,
                          xIN_valve := fb_gripperSolerohrRight.xOUT_VALVE,
                          tIN_GS_ms := 300,  //ms
                          tIN_AS_ms := 300); //ms

// Force control
fb_kraftLeft();
fb_kraftRight();

(*******************************************************************)
(* OUTPUTS *)
(*******************************************************************)
// Error Flag 
xOUT_ErrFlag := (bOUT_Error <> 0) OR (ST125_Pnp_e.ERROR = iOUT_Step);
// Baustein befindet sich im Ablauf 
xOUT_Busy := (iOUT_Step > ST125_Pnp_e.READY) AND (iOUT_Step < ST125_Pnp_e.DONE);
// Baustein hat den Ablauf beendet
xOUT_Done := (iOUT_Step = ST125_Pnp_e.DONE);
// Process ready
xOUT_Ready := (iOUT_Step = ST125_Pnp_e.READY) OR (iOUT_Step = ST125_Pnp_e.waitOnMover);
// Timeout FB 				 		
xOUT_Timeout := TON_Timeout.Q;
// Itialisierung fertig			
xOUT_InitDone := (iOUT_Step = ST125_Pnp_e.READY) OR
                 (iOUT_Step = ST125_Pnp_e.waitOnMover);

// Aktueller Schritt			
iOUT_Step := iOUT_Step; //Im Ablauf gesetzt		
sOUT_Step := TO_STRING(iOUT_Step);
//Fehlernummer	 
bOUT_Error := bOUT_Error; //Im Ablauf/FB gesetzt	
(* Warte (alle Schritte wo auf FG oder Teile gewartet wird) *)
xOUT_Wait := (iOUT_Step = ST125_Pnp_e.DONE) OR
             (iOUT_Step = ST125_Pnp_e.READY) OR
             (iOUT_Step = ST125_Pnp_e.START) OR
             (iOUT_Step = ST125_Pnp_e.waitOnMover) OR
             (iOUT_Step = ST125_Pnp_e.SYNC_MOVER_LEAVE) OR
             (iOUT_Step = ST125_Pnp_e.PnP_WaitOnFeeder);

xOUT_MoverFree := iOUT_Step >= ST125_Pnp_e.MOVER_FREE_OP AND iOUT_Step < ST125_Pnp_e.MOVER_NEEDED_OP;

iOUT_ProcessCompletion := F_GetPercent_2(iAktStep,
                                         ST125_Pnp_e.Pnp_Hor_ToRotTablePos,
                                         ST125_Pnp_e.Pnp_Hor_ToTrackPos,
                                         ST125_Pnp_e.Pnp_HandlingDown,
                                         ST125_Pnp_e.SYNC_MOVER_LEAVE);

xOUT_PickPiece := iOUT_Step = ST125_Pnp_e.Pnp_Hor_ToTrackPos;

IO_BOX.Q5206_14_ST125_greifer_filterhut_links :=
    fb_gripperFilterhutLeft.xOUT_VALVE AND NOT (PNP_SIMULATION AND CONST.USE_SIMULATION);

IO_BOX.Q5207_14_ST125_greifer_filterhut_rechts :=
    fb_gripperFilterhutRight.xOUT_VALVE AND NOT (PNP_SIMULATION AND CONST.USE_SIMULATION);

IO_BOX.Q5208_14_ST125_handling_solerohr_links :=
    fb_handlingSolerohrLeft.xOUT_VALVE AND NOT (PNP_SIMULATION AND CONST.USE_SIMULATION);

IO_BOX.Q5209_14_ST125_handling_solerohr_rechts :=
    fb_handlingSolerohrRight.xOUT_VALVE AND NOT (PNP_SIMULATION AND CONST.USE_SIMULATION);

IO_BOX.Q5210_14_ST125_greifer_solerohr_links :=
    fb_gripperSolerohrLeft.xOUT_VALVE AND NOT (PNP_SIMULATION AND CONST.USE_SIMULATION);

IO_BOX.Q5211_14_ST125_greifer_solerohr_rechts :=
    fb_gripperSolerohrRight.xOUT_VALVE AND NOT (PNP_SIMULATION AND CONST.USE_SIMULATION);

IF 0 = bOUT_Error THEN
    IF fb_axis125_01Y.xOUT_ErrFlag THEN
        bOUT_Error := ST125_Alarm_e.Axis_120_01Y_error;
    ELSIF fb_axis125_02Z.xOUT_ErrFlag THEN
        bOUT_Error := ST125_Alarm_e.Axis_120_02Z_error;
    ELSIF fb_gripperFilterhutLeft.xOUT_ErrFlag THEN
        bOUT_Error := ST125_Alarm_e.Cylinder_griper_filterhut_left;
    ELSIF fb_gripperFilterhutRight.xOUT_ErrFlag THEN
        bOUT_Error := ST125_Alarm_e.Cylinder_griper_filterhut_right;
    ELSIF fb_handlingSolerohrLeft.xOUT_ErrFlag THEN
        bOUT_Error := ST125_Alarm_e.Cylinder_handling_solerohr_left;
    ELSIF fb_handlingSolerohrRight.xOUT_ErrFlag THEN
        bOUT_Error := ST125_Alarm_e.Cylinder_handling_solerohr_right;
    ELSIF fb_gripperSolerohrLeft.xOUT_ErrFlag THEN
        bOUT_Error := ST125_Alarm_e.Cylinder_griper_solerohr_left;
    ELSIF fb_gripperSolerohrRight.xOUT_ErrFlag THEN
        bOUT_Error := ST125_Alarm_e.Cylinder_griper_solerohr_right;
    END_IF
ELSIF iOUT_Step < ST125_Pnp_e.ERROR THEN
    iPreStep  := iOUT_Step;
    iOUT_Step := ST125_Pnp_e.ERROR;
END_IF

(*******************************************************************)
(* Ablauf *)
(*******************************************************************)

(* Sperren *)
IF xIN_Sperre THEN
    iPreStep  := ST125_Pnp_e.RESET;
    iOUT_Step := ST125_Pnp_e.RESET;
    RETURN;
END_IF;

(* Schritt Merker *)
IF iAktStep <> iOUT_Step THEN
    iLastStep := iAktStep;
    iAktStep  := iOUT_Step;
END_IF

(* START *)
rtSTART(CLK := xIN_Start);

(*******************************************************************)
(* Schrittkette  *)
(*******************************************************************)
CASE iOUT_Step OF

(***** RESET *****)
ST125_Pnp_e.RESET: (* Schritt 0-99 *)
    //Initialisierungen
    //Start Init Ablauf
    IF xIN_Init THEN
        iOUT_Step := ST125_Pnp_e.INIT;
        //Start Manu Ablauf
    ELSIF enIN_State = StateMANU AND xIN_NextStep THEN
        iOUT_Step := ST125_Pnp_e.INIT;
    END_IF;

(***** INIT *****)
ST125_Pnp_e.INIT: (* Grundstellung ? *)
    IF fb_axis125_01Y.xOUT_HOMED THEN
        iOUT_Step := ST125_Pnp_e.Init_VerticalsUp;
    ELSE
        iOUT_Step := ST125_Pnp_e.Init_HomeVerticals;
    END_IF;

ST125_Pnp_e.Init_HomeVerticals:
    IF fb_axis125_02Z.xOUT_HOMED THEN
        iOUT_Step := ST125_Pnp_e.Init_VerticalsUp;
    END_IF

ST125_Pnp_e.Init_VerticalsUp:
    IF fb_gripperFilterhutLeft.xIN_AS OR fb_gripperFilterhutRight.xIN_AS THEN
        IF fb_PnpVerAxis.MoveTo(ST125_PnpVerPos_e.UpFull).xOUT_InPos THEN
            IF fb_axis125_01Y.xOUT_READY OR fb_axis125_01Y.xOUT_HOMED THEN
                iOUT_Step := ST125_Pnp_e.Init_HorizontalsToTrack;
            ELSE
                iOUT_Step := ST125_Pnp_e.Init_HomeHorizontals;
            END_IF
        END_IF
    ELSE
        IF fb_PnpVerAxis.MoveTo(ST125_PnpVerPos_e.UpEmpty).xOUT_InPos THEN
            IF fb_axis125_01Y.xOUT_READY OR fb_axis125_01Y.xOUT_HOMED THEN
                iOUT_Step := ST125_Pnp_e.Init_HorizontalsToTrack;
            ELSE
                iOUT_Step := ST125_Pnp_e.Init_HomeHorizontals;
            END_IF
        END_IF
    END_IF

ST125_Pnp_e.Init_HomeHorizontals:
    IF fb_axis125_01Y.xOUT_HOMED THEN
        iOUT_Step := ST125_Pnp_e.Init_HorizontalsToTrack;
    END_IF

ST125_Pnp_e.Init_HorizontalsToTrack:
    IF fb_PnpHorAxis.MoveTo(ST125_PnpHorPos_e.GS).xOUT_InPos THEN
        iOUT_Step := ST125_Pnp_e.Init_open_solenohr_gripper;
    END_IF

ST125_Pnp_e.Init_open_solenohr_gripper:
    IF fb_gripperSolerohrLeft.xOUT_inGS AND fb_gripperSolerohrRight.xOUT_inGS THEN
        iOUT_Step := ST125_Pnp_e.Init_handling_up;
    END_IF

ST125_Pnp_e.Init_handling_up:
    IF fb_handlingSolerohrLeft.xOUT_inGS AND fb_handlingSolerohrRight.xOUT_inGS THEN
        iOUT_Step := ST125_Pnp_e.Init_adjust_left_clamp;
    END_IF

ST125_Pnp_e.Init_adjust_left_clamp:
    // a piece is in the griper when there is no GS signal
    IF _20_AUTO.recipe.st125.xUseVerLeft THEN
        iOUT_Step := ST125_Pnp_e.Init_adjust_right_clamp;
    ELSE
        iOUT_Step := ST125_Pnp_e.Init_open_left_clamp;
    END_IF

ST125_Pnp_e.Init_open_left_clamp:
    IF fb_gripperFilterhutLeft.xIN_AS THEN
        iOUT_Step := ST125_Pnp_e.Init_adjust_right_clamp;
    END_IF

ST125_Pnp_e.Init_adjust_right_clamp:
    // a piece is in the griper when there is no GS signal
    IF _20_AUTO.recipe.st125.xUseVerRight THEN
        iOUT_Step := ST125_Pnp_e.Init_check_if_pces_handled;
    ELSE
        iOUT_Step := ST125_Pnp_e.Init_open_right_clamp;
    END_IF

ST125_Pnp_e.Init_open_right_clamp:
    IF fb_gripperFilterhutRight.xIN_AS THEN
        iOUT_Step := ST125_Pnp_e.Init_check_if_pces_handled;
    END_IF

ST125_Pnp_e.Init_check_if_pces_handled:
    IF (NOT _20_AUTO.recipe.st125.xUseVerLeft AND
       fb_gripperFilterhutLeft.xIN_GS) OR
       (NOT _20_AUTO.recipe.st125.xUseVerRight AND
       NOT fb_gripperFilterhutRight.xIN_GS) THEN
        // ERROR: a piece is present in an unused gripper
        bOUT_Error := ST125_Alarm_e.Piece_in_unused_griper;
        iOUT_Step  := ST125_Pnp_e.ERROR;

        // if both are open, we don't make further checks
    ELSIF fb_gripperFilterhutLeft.xOUT_inAS AND fb_gripperFilterhutRight.xOUT_inAS THEN
        iOUT_Step := ST125_Pnp_e.READY;

    ELSIF (_20_AUTO.recipe.st125.xUseVerLeft AND fb_gripperFilterhutLeft.xOUT_inGS) AND
          (_20_AUTO.recipe.st125.xUseVerRight AND NOT fb_gripperFilterhutRight.xOUT_inGS) THEN
        // ERROR: A piece is missing in the left griper.
        bOUT_Error := ST125_Alarm_e.Piece_missing_left_griper;
        iOUT_Step  := ST125_Pnp_e.ERROR;

    ELSIF (_20_AUTO.recipe.st125.xUseVerLeft AND NOT fb_gripperFilterhutLeft.xOUT_inGS) AND
          (_20_AUTO.recipe.st125.xUseVerRight AND fb_gripperFilterhutRight.xOUT_inGS) THEN
        // ERROR: A piece is missing in the right griper.
        bOUT_Error := ST125_Alarm_e.Piece_missing_right_griper;
        iOUT_Step  := ST125_Pnp_e.ERROR;

    ELSE
        iOUT_Step := ST125_Pnp_e.waitOnMover;
    END_IF

(***** READY / INIT DONE *****)
ST125_Pnp_e.READY:    (* Start AUTO,END,LEER,STEP *)
    IF xIN_Start THEN //IF rtSTART.Q THEN
        iOUT_Step := ST125_Pnp_e.START;
    END_IF

(***** START  ZYKLISCH *****)
ST125_Pnp_e.START: (*  *)
    IF xIN_NextStep AND pxFG_Freigabe^ THEN
        IF enState.StateLEER = enIN_State THEN
            IF __ISVALIDREF(Mover) THEN
                IF Mover.GetLastStationDone() > 0 THEN
                    iOUT_Step := ST125_Pnp_e.Pnp_Hor_ToRotTablePos;
                ELSE
                    iOUT_Step := ST125_Pnp_e.waitOnMover;
                END_IF
            END_IF
        ELSE
            iOUT_Step := ST125_Pnp_e.Pnp_Hor_ToRotTablePos;
        END_IF
    END_IF;

ST125_Pnp_e.Pnp_Hor_ToRotTablePos:
    IF xIN_NextStep AND fb_PnpHorAxis.MoveTo(ST125_PnpHorPos_e.AS).xOUT_InPos THEN
        iOUT_Step := ST125_Pnp_e.Pnp_WaitOnFeeder;
    END_IF

ST125_Pnp_e.Pnp_WaitOnFeeder:
    IF xIN_PceReadyToPick THEN
        iOUT_Step := ST125_Pnp_e.Pnp_Ver_RotTableDown;
    END_IF

ST125_Pnp_e.Pnp_Ver_RotTableDown:
    IF xIN_NextStep AND fb_PnpVerAxis.MoveTo(ST125_PnpVerPos_e.DownEmpty).xOUT_InPos THEN
        iOUT_Step := ST125_Pnp_e.Pnp_takeTubeCap;
    END_IF;

ST125_Pnp_e.Pnp_takeTubeCap:
    IF xIN_NextStep AND
       (NOT _20_AUTO.recipe.st125.xUseVerLeft OR fb_gripperFilterhutLeft.xOUT_inGS) AND
       (NOT _20_AUTO.recipe.st125.xUseVerRight OR fb_gripperFilterhutRight.xOUT_inGS) THEN
        iOUT_Step := ST125_Pnp_e.Pnp_Ver_RotTableUp;
    END_IF;

ST125_Pnp_e.Pnp_Ver_RotTableUp:
    IF xIN_NextStep AND fb_PnpVerAxis.MoveTo(ST125_PnpVerPos_e.UpFull).xOUT_InPos THEN
        iOUT_Step := ST125_Pnp_e.Pnp_Hor_ToTrackPos;
    END_IF;

ST125_Pnp_e.Pnp_Hor_ToTrackPos:
    IF xIN_NextStep AND fb_PnpHorAxis.MoveTo(ST125_PnpHorPos_e.GS).xOUT_InPos THEN
        iOUT_Step := ST125_Pnp_e.waitOnMover;
    END_IF

ST125_Pnp_e.waitOnMover: (*  *)
    IF xIN_NextStep AND __ISVALIDREF(Mover) OR HMI.bArForceCyclusState[StationList_e.ST125] THEN
        IF Mover.GetLastStationDone() >= INT#125 THEN
            iOUT_Step := ST125_Pnp_e.SYNC_MOVER_LEAVE;
        ELSIF Mover.GetLastStationDone() < INT#105 THEN
            iOUT_Step := ST125_Pnp_e.SYNC_MOVER_LEAVE;
        ELSE
            iOUT_Step := ST125_Pnp_e.Pnp_HandlingDown;
        END_IF
    END_IF;

ST125_Pnp_e.Pnp_HandlingDown:
    IF xIN_NextStep AND
       (NOT _20_AUTO.recipe.st125.xUseVerLeft OR fb_handlingSolerohrLeft.xOUT_inAS) AND
       (NOT _20_AUTO.recipe.st125.xUseVerRight OR fb_handlingSolerohrRight.xOUT_inAS) THEN
        iOUT_Step := ST125_Pnp_e.Pnp_closeTubeGriper;
    END_IF;

ST125_Pnp_e.Pnp_closeTubeGriper:
    IF xIN_NextStep AND
       (NOT _20_AUTO.recipe.st125.xUseVerLeft OR fb_gripperSolerohrLeft.xOUT_inAS) AND
       (NOT _20_AUTO.recipe.st125.xUseVerRight OR fb_gripperSolerohrRight.xOUT_inAS) THEN
        iOUT_Step := ST125_Pnp_e.Pnp_Ver_ShuttleDown;
    END_IF;

ST125_Pnp_e.Pnp_Ver_ShuttleDown:
    fb_PnpVerAxis.MoveTo(ST125_PnpVerPos_e.DownFullQuick);

    IF fb_axis125_02Z.xOUT_DONE THEN
        iOUT_Step := ST125_Pnp_e.Pnp_placeCap;

        IF __ISVALIDREF(Mover) THEN
            IF NOT Mover.SetLastStation(125) THEN
                ASSERT(0);
            END_IF
        END_IF
    END_IF

ST125_Pnp_e.Pnp_placeCap:
    IF xIN_NextStep AND
       (NOT _20_AUTO.recipe.st125.xUseVerLeft OR fb_gripperFilterhutLeft.xOUT_inAS) AND
       (NOT _20_AUTO.recipe.st125.xUseVerRight OR fb_gripperFilterhutRight.xOUT_inAS) THEN
        iOUT_Step := ST125_Pnp_e.Pnp_Ver_pushCapTorqueControl;
    END_IF;

ST125_Pnp_e.Pnp_Ver_pushCapTorqueControl:
    IF (fb_PnpVerAxis.MoveTo(ST125_PnpVerPos_e.DownFullTorqueControl).xOUT_InPos OR
        NOT _20_AUTO.recipe.st110.xUseVerLeft) THEN
        IF (PNP_SIMULATION AND CONST.USE_SIMULATION) OR PNP_DONT_CHECK_KRAFT THEN
            iOUT_Step := ST125_Pnp_e.PnP_Ver_quick_stop;
        ELSE
            iOUT_Step := ST125_Pnp_e.ERROR;

        END_IF

    ELSIF fb_kraftLeft.lrOUT_value >= _20_AUTO.recipe.st125.kraft_left_raw OR
          fb_kraftRight.lrOUT_value >= _20_AUTO.recipe.st125.kraft_right_raw THEN
        iOUT_Step := ST125_Pnp_e.PnP_Ver_quick_stop;
    END_IF;

ST125_Pnp_e.PnP_Ver_quick_stop:
    IF xIN_NextStep THEN
        iOUT_Step := ST125_Pnp_e.Pnp_HandlingSolerohrRelease;
    END_IF;

ST125_Pnp_e.Pnp_HandlingSolerohrRelease:
    IF xIN_NextStep AND
       (NOT _20_AUTO.recipe.st125.xUseVerLeft OR fb_gripperSolerohrLeft.xOUT_inGS) AND
       (NOT _20_AUTO.recipe.st125.xUseVerRight OR fb_gripperSolerohrRight.xOUT_inGS) AND
       NOT fb_axis125_02Z.xOUT_BUSY THEN
        iOUT_Step := ST125_Pnp_e.Pnp_Ver_ShuttleFullUp;
    END_IF;

ST125_Pnp_e.Pnp_Ver_ShuttleFullUp:
    IF xIN_NextStep AND fb_PnpVerAxis.MoveTo(ST125_PnpVerPos_e.UpEmpty).xOUT_InPos THEN
        iOUT_Step := ST125_Pnp_e.Pnp_HandlingUp;
    END_IF;

ST125_Pnp_e.Pnp_HandlingUp:
    IF xIN_NextStep AND
       (NOT _20_AUTO.recipe.st125.xUseVerLeft OR fb_handlingSolerohrLeft.xOUT_inGS) AND
       (NOT _20_AUTO.recipe.st125.xUseVerRight OR fb_handlingSolerohrRight.xOUT_inGS) THEN
        iOUT_Step := ST125_Pnp_e.SYNC_MOVER_LEAVE;

        IF __ISVALIDREF(Mover) THEN
            IF NOT Mover.SetLastStation(125) THEN
                ASSERT(0);
            END_IF
        END_IF
    END_IF;

ST125_Pnp_e.SYNC_MOVER_LEAVE:
    // The mover needs to be taken by MoverMan
    IF NOT __ISVALIDREF(Mover) THEN
        IF (NOT _20_AUTO.recipe.st125.xUseVerLeft OR fb_gripperFilterhutLeft.xOUT_inAS) AND
           (NOT _20_AUTO.recipe.st125.xUseVerRight OR fb_gripperFilterhutRight.xOUT_inAS) THEN
            iOUT_Step := ST125_Pnp_e.DONE;
        ELSE
            iOUT_Step := ST125_Pnp_e.waitOnMover;
        END_IF
    END_IF

(***** DONE *****)
ST125_Pnp_e.DONE: (* Letzter Schritt  *)
    IF NOT xIN_AlarmAktiv THEN
        //AUTO
        IF (enIN_State = StateAUTO) AND xIN_RestartCYCL THEN
            iOUT_Step := ST125_Pnp_e.START;
            //STEP / END / LEERFAHREN restart
        ELSIF (enIN_State < StateAUTO) AND (enIN_State >= enState.StateSTEP) AND xIN_RestartCYCL THEN
            iOUT_Step := ST125_Pnp_e.START;
            //STEP / END / LEERFAHREN fertig
        ELSIF (enIN_State = StateREADY) THEN
            iOUT_Step := ST125_Pnp_e.READY;
        END_IF;
    END_IF;

(************ ERROR *************)
ST125_Pnp_e.ERROR: (* ERROR *) ;

END_CASE;

END_FUNCTION_BLOCK

// ---- POUs/20_AUTO/ST125/FB_ABL_125_Feeder.TcPOU
FUNCTION_BLOCK FB_ABL_125_Feeder
(****************************************************************************************)
(*	TITEL				RFID-Ring laden, Feeder and rotary table                        *)
(*	Status				ungetestet                         								*)
(*	Beschrieb:			Ablaufbeschreibung												*)
(*																						*)
(*	Steps:	self-explained using enum													*)
(***********************************Revisionen*******************************************)
(*	see github blames																	*)
(****************************************************************************************)
VAR_INPUT
    xIN_Reset       : BOOL;          // Schrittkette zurücksetzen 
    xIN_Init        : BOOL;          // Initialisieren
    xIN_Quit        : BOOL;          // Fehler quittieren 
    xIN_Start       : BOOL;          // Startbefehl
    xIN_Sperre      : BOOL;          // FB Sperren 
    xIN_NextStep    : BOOL;          // Nächsten Schritt ausführen 
    xIN_AlarmAktiv  : BOOL;          // Anlage hat Alarm
    xIN_DryCycle    : BOOL;          // Fahren ohne Teile
    xIN_RestartCYCL : BOOL;          // Zyklus erneut starten im STEP, END, LEERFAHREN
    enIN_State      : enState;       // Status Anlage
    tIN_Timeout     : TIME := T#10s; // Timout

    pxFG_Freigabe : POINTER TO BOOL; //Freigabe von Station

